C03568=1021.069,418.484,-159.354,174.058,50.310,160.418
C03569=1021.080,418.730,-159.402,174.072,50.312,160.420
C03570=1021.092,418.975,-159.450,174.087,50.313,160.423
C03571=1021.104,419.220,-159.498,174.100,50.315,160.426
C03572=1021.115,419.465,-159.546,174.115,50.316,160.429
C03573=1021.127,419.710,-159.594,174.129,50.318,160.432
C03574=1021.139,419.955,-159.641,174.143,50.320,160.435
C03575=1021.150,420.201,-159.690,174.158,50.321,160.438
C03576=1021.161,420.446,-159.737,174.171,50.323,160.441
C03577=1021.173,420.691,-159.786,174.186,50.325,160.444
C03578=1021.185,420.936,-159.834,174.201,50.326,160.446
C03579=1021.197,421.181,-159.882,174.215,50.328,160.449
C03580=1021.208,421.427,-159.930,174.229,50.330,160.453
C03581=1021.220,421.671,-159.979,174.244,50.331,160.455
C03582=1021.231,421.916,-160.027,174.259,50.333,160.458
C03583=1021.243,422.161,-160.076,174.273,50.335,160.461
C03584=1021.255,422.406,-160.125,174.287,50.337,160.464
C03585=1021.267,422.652,-160.173,174.302,50.338,160.467
C03586=1021.279,422.896,-160.222,174.317,50.340,160.471
C03587=1021.290,423.141,-160.271,174.332,50.342,160.474
C03588=1021.302,423.386,-160.320,174.347,50.344,160.477
C03589=1021.314,423.631,-160.368,174.362,50.346,160.480
C03590=1021.326,423.877,-160.417,174.377,50.348,160.483
C03591=1021.338,424.121,-160.466,174.392,50.349,160.486
C03592=1021.350,424.365,-160.515,174.407,50.351,160.489
C03593=1021.363,424.610,-160.564,174.422,50.354,160.492
C03594=1021.375,424.856,-160.613,174.437,50.355,160.495
C03595=1021.386,425.101,-160.662,174.452,50.358,160.499
C03596=1021.399,425.346,-160.711,174.467,50.359,160.502
C03597=1021.411,425.591,-160.761,174.482,50.362,160.505
C03598=1021.423,425.835,-160.810,174.498,50.363,160.508
C03599=1021.435,426.081,-160.860,174.513,50.365,160.511
C03600=1021.446,426.325,-160.909,174.529,50.367,160.515
C03601=1021.459,426.570,-160.958,174.544,50.370,160.518
C03602=1021.471,426.810,-161.007,174.559,50.371,160.521
C03603=1021.483,427.050,-161.056,174.574,50.374,160.524
C03604=1021.495,427.290,-161.104,174.589,50.376,160.528
C03605=1021.507,427.530,-161.153,174.605,50.378,160.531
C03606=1021.519,427.770,-161.202,174.620,50.379,160.534
C03607=1021.531,428.009,-161.252,174.636,50.382,160.537
C03608=1021.544,428.249,-161.300,174.651,50.384,160.541
C03609=1021.555,428.488,-161.349,174.666,50.386,160.544
C03610=1021.567,428.733,-161.399,174.682,50.388,160.547
C03611=1021.580,428.978,-161.449,174.698,50.391,160.551
C03612=1021.592,429.223,-161.499,174.714,50.393,160.554
C03613=1021.605,429.467,-161.549,174.730,50.395,160.557
C03614=1021.618,429.712,-161.599,174.746,50.397,160.561
C03615=1021.630,429.956,-161.649,174.762,50.399,160.564
C03616=1021.643,430.202,-161.700,174.778,50.402,160.568
C03617=1021.655,430.446,-161.751,174.795,50.404,160.571
C03618=1021.272,428.491,-161.685,174.655,50.455,160.562
C03619=1021.261,428.264,-161.639,174.641,50.453,160.559
C03620=1021.250,428.037,-161.592,174.626,50.451,160.556
C03621=1021.238,427.810,-161.547,174.611,50.449,160.553
C03622=1021.227,427.582,-161.500,174.597,50.447,160.550
C03623=1021.216,427.356,-161.454,174.582,50.445,160.547
C03624=1021.204,427.128,-161.408,174.567,50.444,160.544
C03625=1021.193,426.901,-161.361,174.553,50.442,160.541
C03626=1021.182,426.673,-161.315,174.539,50.440,160.538
C03627=1021.169,426.429,-161.267,174.523,50.438,160.534
C03628=1021.157,426.184,-161.216,174.508,50.436,160.531
C03629=1021.146,425.939,-161.167,174.492,50.434,160.528
C03630=1021.133,425.695,-161.117,174.477,50.432,160.525
C03631=1021.121,425.449,-161.068,174.462,50.430,160.522
C03632=1021.109,425.205,-161.020,174.447,50.428,160.518
C03633=1021.097,424.959,-160.970,174.431,50.426,160.515
C03634=1021.085,424.714,-160.921,174.416,50.425,160.512
C03635=1021.073,424.470,-160.872,174.401,50.423,160.509
C03636=1021.061,424.224,-160.822,174.386,50.421,160.506
C03637=1021.049,423.980,-160.774,174.371,50.419,160.503
C03638=1021.037,423.735,-160.724,174.356,50.417,160.500
C03639=1021.025,423.490,-160.677,174.341,50.416,160.496
C03640=1021.013,423.245,-160.628,174.326,50.414,160.493
C03641=1021.001,422.999,-160.578,174.311,50.412,160.490
C03642=1020.989,422.755,-160.530,174.297,50.410,160.487
C03643=1020.978,422.510,-160.481,174.282,50.409,160.484
C03644=1020.966,422.265,-160.433,174.267,50.407,160.481
C03645=1020.954,422.020,-160.384,174.252,50.406,160.478
C03646=1020.942,421.775,-160.336,174.237,50.404,160.475
C03647=1020.931,421.530,-160.287,174.223,50.402,160.472
C03648=1020.920,421.285,-160.239,174.209,50.400,160.469
C03649=1020.907,421.040,-160.190,174.194,50.399,160.466
C03650=1020.895,420.794,-160.142,174.179,50.397,160.463
C03651=1020.884,420.549,-160.094,174.165,50.396,160.460
C03652=1020.872,420.304,-160.046,174.150,50.395,160.458
C03653=1020.861,420.059,-159.998,174.136,50.393,160.455
C03654=1020.849,419.814,-159.950,174.122,50.391,160.452
C03655=1020.837,419.569,-159.902,174.108,50.390,160.449
C03656=1020.826,419.324,-159.854,174.094,50.388,160.446
C03657=1020.814,419.079,-159.806,174.079,50.387,160.443
C03658=1020.803,418.833,-159.759,174.065,50.386,160.440
C03659=1020.791,418.588,-159.711,174.051,50.384,160.437
C03660=1020.780,418.343,-159.663,174.037,50.383,160.435
C03661=1020.768,418.098,-159.616,174.023,50.381,160.432
C03662=1020.757,417.853,-159.567,174.009,50.380,160.429
C03663=1020.746,417.607,-159.520,173.995,50.378,160.426
C03664=1020.734,417.362,-159.473,173.981,50.377,160.423
C03665=1020.723,417.117,-159.425,173.967,50.376,160.421
C03666=1020.712,416.872,-159.378,173.954,50.374,160.418
C03667=1020.701,416.626,-159.329,173.940,50.373,160.415
C03668=1020.690,416.381,-159.283,173.926,50.372,160.412
C03669=1020.678,416.136,-159.235,173.913,50.370,160.410
C03670=1020.667,415.890,-159.187,173.898,50.369,160.407
C03671=1020.656,415.645,-159.141,173.885,50.368,160.404
C03672=1020.644,415.400,-159.093,173.872,50.366,160.401
C03673=1020.634,415.155,-159.046,173.858,50.365,160.399
C03674=1020.623,414.909,-158.999,173.844,50.364,160.396
C03675=1020.612,414.664,-158.952,173.831,50.363,160.394
C03676=1020.600,414.419,-158.905,173.818,50.362,160.391
C03677=1020.589,414.174,-158.859,173.803,50.360,160.388
C03678=1020.578,413.928,-158.812,173.790,50.359,160.386
C03679=1020.568,413.683,-158.765,173.777,50.358,160.383
C03680=1020.556,413.437,-158.718,173.764,50.357,160.381
C03681=1020.545,413.192,-158.672,173.751,50.356,160.378
C03682=1020.535,412.947,-158.625,173.738,50.355,160.375
C03683=1020.519,412.599,-158.559,173.719,50.353,160.372
C03684=1020.503,412.251,-158.493,173.700,50.352,160.368
C03685=1020.488,411.903,-158.427,173.682,50.351,160.365
C03686=1020.472,411.556,-158.361,173.663,50.349,160.361
C03687=1020.461,411.311,-158.315,173.651,50.348,160.359
C03688=1020.451,411.065,-158.269,173.637,50.347,160.356
C03689=1020.440,410.820,-158.223,173.624,50.346,160.353
C03690=1020.430,410.574,-158.176,173.611,50.345,160.351
C03691=1020.419,410.329,-158.130,173.599,50.344,160.349
C03692=1020.409,410.083,-158.084,173.586,50.343,160.346
C03693=1020.398,409.838,-158.037,173.573,50.342,160.344
C03694=1020.387,409.592,-157.991,173.561,50.341,160.341
C03695=1020.376,409.347,-157.945,173.548,50.340,160.339
C03696=1020.366,409.101,-157.900,173.535,50.340,160.336
C03697=1020.355,408.856,-157.854,173.523,50.338,160.334
C03698=1020.345,408.610,-157.808,173.510,50.338,160.332
C03699=1020.334,408.365,-157.762,173.497,50.337,160.329
C03700=1020.323,408.119,-157.716,173.484,50.336,160.327
C03701=1020.312,407.873,-157.671,173.473,50.335,160.324
C03702=1020.302,407.627,-157.625,173.460,50.335,160.322
C03703=1020.291,407.382,-157.579,173.447,50.334,160.320
C03704=1020.281,407.137,-157.534,173.434,50.334,160.317
C03705=1020.271,406.891,-157.489,173.423,50.333,160.315
C03706=1020.259,406.645,-157.443,173.410,50.332,160.313
C03707=1020.249,406.399,-157.398,173.398,50.331,160.311
C03708=1020.239,406.154,-157.353,173.386,50.331,160.308
C03709=1020.229,405.908,-157.308,173.373,50.330,160.306
C03710=1020.217,405.663,-157.262,173.361,50.329,160.304
C03711=1020.208,405.417,-157.217,173.349,50.329,160.301
C03712=1020.197,405.172,-157.171,173.337,50.328,160.299
C03713=1020.187,404.926,-157.127,173.324,50.327,160.297
C03714=1020.177,404.680,-157.081,173.313,50.327,160.295
C03715=1020.166,404.435,-157.037,173.300,50.326,160.292
C03716=1020.156,404.189,-156.991,173.288,50.325,160.290
C03717=1020.146,403.944,-156.947,173.276,50.325,160.288
C03718=1020.136,403.697,-156.901,173.264,50.324,160.286
C03719=1020.125,403.452,-156.857,173.253,50.324,160.284
C03720=1020.115,403.206,-156.812,173.240,50.323,160.281
C03721=1020.105,402.961,-156.767,173.229,50.323,160.279
C03722=1020.096,402.715,-156.722,173.216,50.323,160.277
C03723=1020.085,402.469,-156.677,173.205,50.322,160.275
C03724=1020.075,402.224,-156.633,173.193,50.321,160.273
C03725=1020.065,401.978,-156.588,173.181,50.321,160.271
C03726=1020.055,401.733,-156.543,173.169,50.320,160.268
C03727=1020.045,401.486,-156.498,173.158,50.320,160.266
C03728=1020.035,401.241,-156.454,173.147,50.320,160.264
C03729=1020.025,400.995,-156.410,173.134,50.320,160.262
C03730=1020.016,400.750,-156.365,173.123,50.319,160.260
C03731=1020.006,400.503,-156.321,173.111,50.318,160.258
C03732=1019.995,400.257,-156.276,173.100,50.318,160.256
C03733=1019.986,400.011,-156.232,173.088,50.318,160.254
C03734=1019.976,399.766,-156.187,173.076,50.318,160.252
C03735=1019.966,399.520,-156.144,173.065,50.317,160.250
C03736=1019.956,399.275,-156.099,173.054,50.317,160.248
C03737=1019.946,399.029,-156.055,173.042,50.316,160.246
C03738=1019.937,398.783,-156.011,173.031,50.316,160.244
C03739=1019.927,398.537,-155.966,173.020,50.316,160.242
C03740=1019.917,398.291,-155.923,173.008,50.316,160.240
C03741=1019.907,398.045,-155.879,172.997,50.316,160.238
C03742=1019.897,397.799,-155.835,172.985,50.316,160.236
C03743=1019.885,397.475,-155.777,172.971,50.316,160.233
C03744=1019.872,397.150,-155.720,172.955,50.315,160.231
C03745=1019.858,396.825,-155.662,172.941,50.315,160.228
C03746=1019.846,396.500,-155.604,172.926,50.315,160.226
C03747=1019.836,396.254,-155.560,172.915,50.315,160.224
C03748=1019.826,396.009,-155.517,172.904,50.315,160.222
C03749=1019.816,395.762,-155.473,172.892,50.315,160.220
C03750=1019.807,395.516,-155.430,172.882,50.315,160.218
C03751=1019.798,395.271,-155.386,172.871,50.314,160.216
C03752=1019.788,395.025,-155.343,172.860,50.314,160.214
C03753=1019.777,394.779,-155.299,172.849,50.315,160.212
C03754=1019.768,394.532,-155.256,172.838,50.315,160.211
C03755=1019.759,394.287,-155.213,172.827,50.314,160.208
C03756=1019.749,394.041,-155.170,172.816,50.314,160.207
C03757=1019.740,393.794,-155.126,172.805,50.315,160.205
C03758=1019.730,393.549,-155.083,172.794,50.315,160.203
C03759=1019.721,393.303,-155.039,172.783,50.315,160.201
C03760=1019.711,393.056,-154.997,172.773,50.315,160.200
C03761=1019.702,392.810,-154.954,172.763,50.315,160.198
C03762=1019.692,392.564,-154.910,172.751,50.315,160.196
C03763=1019.683,392.318,-154.868,172.740,50.315,160.194
C03764=1019.673,392.072,-154.825,172.730,50.316,160.192
C03765=1019.664,391.826,-154.782,172.720,50.315,160.191
C03766=1019.655,391.580,-154.739,172.709,50.316,160.189
C03767=1019.645,391.334,-154.696,172.698,50.316,160.187
C03768=1019.636,391.088,-154.653,172.687,50.316,160.185
C03769=1019.626,390.842,-154.611,172.677,50.316,160.183
C03770=1019.616,390.596,-154.568,172.667,50.317,160.182
C03771=1019.608,390.350,-154.525,172.656,50.317,160.180
C03772=1019.599,390.103,-154.483,172.645,50.317,160.178
C03773=1019.589,389.857,-154.440,172.635,50.317,160.177
C03774=1019.580,389.611,-154.398,172.624,50.318,160.175
C03775=1019.571,389.365,-154.355,172.614,50.317,160.173
C03776=1019.562,389.119,-154.312,172.604,50.318,160.171
C03777=1019.552,388.873,-154.270,172.593,50.318,160.170
C03778=1019.543,388.627,-154.228,172.583,50.319,160.168
C03779=1019.534,388.380,-154.185,172.572,50.319,160.166
C03780=1019.524,388.134,-154.143,172.562,50.320,160.165
C03781=1019.515,387.888,-154.101,172.552,50.319,160.163
C03782=1019.506,387.642,-154.058,172.541,50.320,160.161
C03783=1019.497,387.395,-154.016,172.532,50.321,160.160
C03784=1019.488,387.149,-153.973,172.521,50.321,160.158
C03785=1019.479,386.903,-153.932,172.511,50.321,160.156
C03786=1019.470,386.656,-153.890,172.501,50.322,160.155
C03787=1019.461,386.411,-153.847,172.490,50.323,160.153
C03788=1019.452,386.164,-153.806,172.481,50.323,160.152
C03789=1019.443,385.918,-153.764,172.470,50.323,160.150
C03790=1019.434,385.672,-153.722,172.460,50.324,160.148
C03791=1019.425,385.426,-153.680,172.451,50.324,160.147
C03792=1019.416,385.179,-153.638,172.440,50.325,160.145
C03793=1019.407,384.932,-153.596,172.431,50.325,160.144
C03794=1019.397,384.686,-153.555,172.420,50.326,160.142
C03795=1019.388,384.440,-153.513,172.410,50.326,160.141
C03796=1019.379,384.194,-153.472,172.400,50.327,160.139
C03797=1019.370,383.947,-153.430,172.391,50.328,160.138
C03798=1019.361,383.701,-153.388,172.380,50.329,160.136
C03799=1019.351,383.455,-153.347,172.371,50.329,160.135
C03800=1019.343,383.209,-153.306,172.360,50.330,160.133
C03801=1019.335,382.962,-153.265,172.351,50.330,160.132
C03802=1019.326,382.716,-153.223,172.341,50.331,160.130
C03803=1019.314,382.429,-153.174,172.329,50.332,160.128
C03804=1019.304,382.141,-153.127,172.318,50.333,160.127
C03805=1019.294,381.854,-153.079,172.306,50.334,160.125
C03806=1019.283,381.567,-153.030,172.296,50.335,160.123
C03807=1019.275,381.321,-152.989,172.285,50.336,160.122
C03808=1019.266,381.074,-152.948,172.276,50.336,160.120
C03809=1019.257,380.828,-152.906,172.267,50.337,160.119
C03810=1019.248,380.581,-152.865,172.256,50.338,160.117
C03811=1019.239,380.335,-152.824,172.247,50.339,160.116
C03812=1019.231,380.088,-152.783,172.238,50.340,160.115
C03813=1019.222,379.841,-152.742,172.228,50.340,160.113
C03814=1019.214,379.596,-152.701,172.218,50.341,160.112
C03815=1019.205,379.349,-152.660,172.208,50.342,160.110
C03816=1019.196,379.102,-152.620,172.199,50.343,160.109
C03817=1019.188,378.857,-152.578,172.190,50.344,160.108
C03818=1019.179,378.610,-152.537,172.180,50.344,160.106
C03819=1019.171,378.363,-152.497,172.170,50.345,160.105
C03820=1019.162,378.117,-152.455,172.161,50.346,160.103
C03821=1019.153,377.871,-152.415,172.152,50.347,160.102
C03822=1019.145,377.624,-152.374,172.143,50.348,160.101
C03823=1019.137,377.378,-152.333,172.133,50.349,160.099
C03824=1019.128,377.131,-152.292,172.123,50.350,160.098
C03825=1019.119,376.885,-152.252,172.114,50.351,160.097
C03826=1019.110,376.638,-152.211,172.105,50.352,160.095
C03827=1019.102,376.391,-152.170,172.096,50.353,160.094
C03828=1019.094,376.144,-152.129,172.087,50.354,160.093
C03829=1019.086,375.898,-152.089,172.077,50.355,160.091
C03830=1019.076,375.651,-152.048,172.068,50.356,160.090
C03831=1019.068,375.405,-152.008,172.059,50.357,160.089
C03832=1019.060,375.159,-151.968,172.050,50.358,160.087
C03833=1019.051,374.912,-151.928,172.040,50.359,160.086
C03834=1019.043,374.666,-151.887,172.031,50.361,160.085
C03835=1019.034,374.418,-151.848,172.022,50.362,160.084
C03836=1019.025,374.172,-151.807,172.013,50.363,160.082
C03837=1019.017,373.925,-151.768,172.003,50.364,160.081
C03838=1019.009,373.679,-151.727,171.995,50.365,160.080
C03839=1019.000,373.432,-151.687,171.986,50.366,160.079
C03840=1018.991,373.186,-151.647,171.976,50.367,160.077
C03841=1018.983,372.939,-151.608,171.968,50.369,160.076
C03842=1018.974,372.692,-151.567,171.958,50.370,160.075
C03843=1018.966,372.445,-151.527,171.950,50.372,160.074
C03844=1018.958,372.199,-151.487,171.940,50.372,160.072
C03845=1018.950,371.953,-151.447,171.932,50.374,160.071
C03846=1018.941,371.706,-151.408,171.923,50.375,160.070
C03847=1018.933,371.460,-151.367,171.914,50.377,160.069
C03848=1018.924,371.212,-151.328,171.905,50.378,160.068
C03849=1018.916,370.966,-151.288,171.896,50.379,160.067
C03850=1018.908,370.719,-151.248,171.887,50.380,160.065
C03851=1018.899,370.473,-151.208,171.878,50.382,160.064
C03852=1018.892,370.226,-151.168,171.869,50.383,160.063
C03853=1018.883,369.979,-151.129,171.860,50.384,160.062
C03854=1018.876,369.732,-151.089,171.851,50.386,160.061
C03855=1018.867,369.486,-151.050,171.842,50.387,160.059
C03856=1018.859,369.239,-151.010,171.834,50.388,160.058
C03857=1018.851,368.992,-150.971,171.825,50.390,160.057
C03858=1018.842,368.746,-150.931,171.817,50.391,160.056
C03859=1018.835,368.499,-150.891,171.808,50.393,160.055
C03860=1018.826,368.252,-150.852,171.799,50.394,160.054
C03861=1018.819,368.005,-150.812,171.790,50.395,160.053
C03862=1018.810,367.759,-150.773,171.781,50.397,160.051
C03863=1018.801,367.494,-150.731,171.772,50.398,160.050
C03864=1018.793,367.229,-150.689,171.763,50.400,160.049
C03865=1018.784,366.963,-150.647,171.754,50.402,160.048
C03866=1018.775,366.699,-150.604,171.745,50.404,160.047
C03867=1018.767,366.452,-150.566,171.736,50.405,160.046
C03868=1018.759,366.205,-150.527,171.727,50.407,160.045
C03869=1018.750,365.958,-150.488,171.719,50.408,160.044
C03870=1018.743,365.712,-150.449,171.710,50.410,160.043
C03871=1018.734,365.465,-150.410,171.701,50.411,160.041
C03872=1018.727,365.218,-150.370,171.693,50.413,160.040
C03873=1018.719,364.971,-150.332,171.685,50.415,160.040
C03874=1018.710,364.724,-150.293,171.676,50.416,160.038
C03875=1018.703,364.477,-150.254,171.667,50.418,160.037
C03876=1018.694,364.230,-150.216,171.659,50.420,160.036
C03877=1018.686,363.984,-150.176,171.651,50.421,160.035
C03878=1018.678,363.737,-150.138,171.642,50.423,160.034
C03879=1018.670,363.490,-150.100,171.634,50.425,160.033
C03880=1018.662,363.243,-150.060,171.625,50.427,160.032
C03881=1018.654,362.997,-150.022,171.617,50.428,160.031
C03882=1018.647,362.749,-149.983,171.609,50.430,160.030
C03883=1018.639,362.502,-149.944,171.600,50.432,160.029
C03884=1018.631,362.256,-149.906,171.591,50.433,160.028
C03885=1018.623,362.009,-149.867,171.584,50.435,160.027
C03886=1018.615,361.762,-149.828,171.575,50.437,160.026
C03887=1018.607,361.515,-149.790,171.567,50.439,160.025
C03888=1018.599,361.268,-149.751,171.560,50.441,160.025
C03889=1018.591,361.022,-149.713,171.551,50.442,160.023
C03890=1018.583,360.774,-149.674,171.542,50.445,160.023
C03891=1018.577,360.563,-149.641,171.536,50.445,160.022
C03892=1018.571,360.352,-149.609,171.528,50.447,160.021
C03893=1018.564,360.142,-149.575,171.522,50.449,160.020
C03894=1018.557,359.931,-149.543,171.514,50.451,160.019
C03895=1018.550,359.720,-149.510,171.508,50.452,160.019
C03896=1018.544,359.509,-149.478,171.501,50.454,160.018
C03897=1018.538,359.299,-149.445,171.494,50.455,160.017
C03898=1018.531,359.088,-149.413,171.487,50.457,160.016
C03899=1018.523,358.841,-149.375,171.478,50.459,160.015
C03900=1018.515,358.595,-149.336,171.471,50.461,160.014
C03901=1018.507,358.347,-149.298,171.462,50.463,160.013
C03902=1018.500,358.100,-149.260,171.455,50.465,160.013
C03903=1018.492,357.853,-149.222,171.446,50.467,160.012
C03904=1018.484,357.606,-149.184,171.438,50.469,160.011
C03905=1018.476,357.360,-149.146,171.431,50.471,160.010
C03906=1018.468,357.112,-149.108,171.422,50.473,160.009
C03907=1018.461,356.865,-149.070,171.414,50.475,160.008
C03908=1018.453,356.618,-149.033,171.406,50.477,160.007
C03909=1018.445,356.371,-148.994,171.398,50.479,160.006
C03910=1018.437,356.124,-148.957,171.391,50.481,160.006
C03911=1018.430,355.877,-148.920,171.382,50.483,160.005
C03912=1018.423,355.631,-148.881,171.374,50.485,160.004
C03913=1018.415,355.383,-148.843,171.366,50.487,160.003
C03914=1018.407,355.136,-148.807,171.358,50.490,160.002
C03915=1018.399,354.889,-148.768,171.351,50.492,160.001
C03916=1018.392,354.642,-148.731,171.343,50.494,160.001
C03917=1018.385,354.395,-148.693,171.335,50.496,160.000
C03918=1018.376,354.148,-148.656,171.327,50.498,159.999
C03919=1018.369,353.900,-148.618,171.320,50.501,159.998
C03920=1018.361,353.654,-148.580,171.311,50.503,159.997
C03921=1018.354,353.407,-148.543,171.304,50.505,159.997
C03922=1018.346,353.160,-148.506,171.296,50.508,159.996
C03923=1018.336,352.830,-148.457,171.286,50.510,159.995
C03924=1018.326,352.500,-148.406,171.275,50.513,159.994
C03925=1018.315,352.170,-148.356,171.265,50.516,159.993
C03926=1018.305,351.840,-148.306,171.255,50.520,159.992
C03927=1018.298,351.592,-148.270,171.246,50.522,159.991
C03928=1018.290,351.346,-148.233,171.239,50.524,159.990
C03929=1018.283,351.098,-148.195,171.231,50.527,159.989
C03930=1018.276,350.851,-148.158,171.224,50.529,159.989
C03931=1018.268,350.604,-148.121,171.216,50.531,159.988
C03932=1018.261,350.357,-148.084,171.209,50.534,159.987
C03933=1018.253,350.110,-148.047,171.200,50.536,159.986
C03934=1018.246,349.863,-148.009,171.193,50.538,159.986
C03935=1018.238,349.616,-147.973,171.185,50.541,159.985
C03936=1018.231,349.368,-147.936,171.178,50.543,159.984
C03937=1018.223,349.121,-147.898,171.171,50.545,159.984
C03938=1018.216,348.874,-147.862,171.163,50.548,159.983
C03939=1018.209,348.627,-147.825,171.156,50.551,159.982
C03940=1018.201,348.380,-147.788,171.147,50.553,159.981
C03941=1018.194,348.133,-147.751,171.140,50.555,159.981
C03942=1018.186,347.886,-147.714,171.132,50.558,159.980
C03943=1018.179,347.638,-147.677,171.125,50.561,159.980
C03944=1018.171,347.391,-147.640,171.118,50.563,159.979
C03945=1018.165,347.144,-147.604,171.110,50.565,159.978
C03946=1018.157,346.897,-147.567,171.103,50.568,159.977
C03947=1018.150,346.650,-147.530,171.095,50.571,159.977
C03948=1018.142,346.402,-147.494,171.088,50.573,159.976
C03949=1018.135,346.155,-147.458,171.080,50.576,159.975
C03950=1018.128,345.908,-147.421,171.073,50.578,159.975
C03951=1018.120,345.661,-147.384,171.066,50.581,159.974
C03952=1018.113,345.413,-147.348,171.058,50.584,159.973
C03953=1018.106,345.166,-147.312,171.051,50.586,159.973
C03954=1018.099,344.919,-147.275,171.043,50.589,159.972
C03955=1018.091,344.672,-147.239,171.036,50.592,159.972
C03956=1018.083,344.425,-147.202,171.029,50.594,159.971
C03957=1018.077,344.178,-147.166,171.021,50.597,159.970
C03958=1018.069,343.930,-147.130,171.014,50.600,159.970
C03959=1018.061,343.683,-147.093,171.006,50.603,159.969
C03960=1018.055,343.436,-147.057,170.999,50.605,159.969
C03961=1018.047,343.188,-147.021,170.992,50.608,159.968
C03962=1018.040,342.941,-146.985,170.984,50.611,159.967
C03963=1018.033,342.694,-146.948,170.977,50.613,159.967
C03964=1018.026,342.446,-146.912,170.970,50.616,159.966
C03965=1018.018,342.199,-146.876,170.963,50.619,159.966
C03966=1018.011,341.951,-146.841,170.956,50.622,159.965
C03967=1018.005,341.704,-146.804,170.949,50.624,159.964
C03968=1017.997,341.457,-146.768,170.941,50.628,159.964
C03969=1017.990,341.210,-146.732,170.934,50.630,159.963
C03970=1017.982,340.963,-146.696,170.927,50.633,159.963
C03971=1017.976,340.715,-146.661,170.920,50.636,159.962
C03972=1017.969,340.468,-146.624,170.913,50.639,159.962
C03973=1017.962,340.221,-146.588,170.906,50.642,159.961
C03974=1017.954,339.973,-146.552,170.898,50.645,159.961
C03975=1017.947,339.726,-146.517,170.891,50.648,159.960
C03976=1017.939,339.479,-146.480,170.884,50.650,159.960
C03977=1017.933,339.231,-146.445,170.877,50.654,159.959
C03978=1017.926,338.984,-146.409,170.870,50.656,159.958
C03979=1017.919,338.737,-146.373,170.863,50.659,159.958
C03980=1017.912,338.489,-146.338,170.855,50.663,159.958
C03981=1017.905,338.241,-146.302,170.848,50.665,159.957
C03982=1017.897,337.995,-146.266,170.842,50.668,159.956
C03983=1017.890,337.735,-146.229,170.834,50.672,159.956
C03984=1017.883,337.474,-146.192,170.826,50.674,159.955
C03985=1017.875,337.214,-146.155,170.819,50.678,159.955
C03986=1017.867,336.953,-146.117,170.812,50.681,159.954
C03987=1017.860,336.706,-146.082,170.805,50.684,159.954
C03988=1017.853,336.459,-146.047,170.798,50.688,159.953
C03989=1017.846,336.211,-146.011,170.791,50.690,159.953
C03990=1017.839,335.964,-145.975,170.784,50.693,159.952
C03991=1017.832,335.717,-145.940,170.776,50.697,159.952
C03992=1017.825,335.469,-145.905,170.770,50.700,159.952
C03993=1017.818,335.221,-145.869,170.763,50.703,159.951
C03994=1017.811,334.974,-145.834,170.756,50.706,159.951
C03995=1017.804,334.727,-145.798,170.749,50.709,159.950
C03996=1017.797,334.480,-145.763,170.742,50.713,159.950
C03997=1017.790,334.232,-145.728,170.736,50.716,159.949
C03998=1017.783,333.984,-145.693,170.729,50.719,159.949
C03999=1017.777,333.737,-145.658,170.721,50.722,159.949
C04000=1017.770,333.490,-145.622,170.715,50.725,159.948
C04001=1017.763,333.242,-145.587,170.708,50.728,159.948
C04002=1017.756,332.995,-145.552,170.702,50.732,159.947
C04003=1017.749,332.747,-145.517,170.694,50.735,159.947
C04004=1017.741,332.500,-145.482,170.687,50.738,159.946
C04005=1017.735,332.252,-145.447,170.681,50.741,159.946
C04006=1017.728,332.005,-145.412,170.674,50.744,159.946
C04007=1017.721,331.757,-145.377,170.666,50.748,159.945
C04008=1017.714,331.510,-145.343,170.660,50.752,159.945
C04009=1017.707,331.263,-145.308,170.654,50.755,159.944
C04010=1017.700,331.015,-145.273,170.647,50.758,159.944
C04011=1017.693,330.768,-145.239,170.639,50.761,159.944
C04012=1017.686,330.520,-145.204,170.633,50.765,159.943
C04013=1017.680,330.273,-145.169,170.626,50.768,159.943
C04014=1017.672,330.025,-145.135,170.620,50.771,159.943
C04015=1017.666,329.778,-145.100,170.613,50.775,159.942
C04016=1017.659,329.530,-145.064,170.606,50.779,159.942
C04017=1017.652,329.282,-145.030,170.599,50.782,159.941
C04018=1017.645,329.035,-144.995,170.593,50.785,159.941
C04019=1017.638,328.787,-144.961,170.586,50.789,159.941
C04020=1017.632,328.540,-144.926,170.579,50.792,159.940
C04021=1017.624,328.292,-144.892,170.573,50.796,159.940
C04022=1017.618,328.045,-144.857,170.566,50.799,159.940
C04023=1017.611,327.797,-144.823,170.560,50.803,159.939
C04024=1017.604,327.550,-144.788,170.552,50.806,159.939
C04025=1017.598,327.303,-144.754,170.546,50.810,159.939
C04026=1017.591,327.055,-144.719,170.539,50.813,159.938
C04027=1017.584,326.808,-144.685,170.533,50.817,159.938
C04028=1017.577,326.560,-144.651,170.526,50.820,159.938
C04029=1017.571,326.312,-144.615,170.519,50.824,159.937
C04030=1017.563,326.065,-144.582,170.513,50.828,159.937
C04031=1017.557,325.818,-144.548,170.506,50.831,159.937
C04032=1017.550,325.570,-144.514,170.500,50.835,159.937
C04033=1017.543,325.322,-144.480,170.493,50.839,159.936
C04034=1017.536,325.075,-144.445,170.487,50.843,159.936
C04035=1017.529,324.827,-144.412,170.480,50.846,159.936
C04036=1017.522,324.579,-144.377,170.474,50.849,159.935
C04037=1017.515,324.332,-144.344,170.467,50.854,159.935
C04038=1017.508,324.085,-144.310,170.460,50.857,159.935
C04039=1017.501,323.837,-144.276,170.454,50.861,159.935
C04040=1017.495,323.589,-144.242,170.448,50.865,159.935
C04041=1017.488,323.342,-144.208,170.441,50.869,159.934
C04042=1017.481,323.094,-144.175,170.434,50.872,159.934
C04043=1017.474,322.829,-144.138,170.427,50.877,159.934
C04044=1017.466,322.565,-144.102,170.421,50.881,159.934
C04045=1017.459,322.300,-144.066,170.414,50.885,159.933
C04046=1017.452,322.035,-144.030,170.407,50.889,159.933
C04047=1017.445,321.788,-143.996,170.400,50.893,159.933
C04048=1017.438,321.540,-143.963,170.394,50.896,159.933
C04049=1017.431,321.292,-143.929,170.388,50.900,159.932
C04050=1017.425,321.045,-143.895,170.381,50.904,159.932
C04051=1017.418,320.798,-143.861,170.375,50.908,159.932
C04052=1017.412,320.550,-143.829,170.368,50.912,159.932
C04053=1017.405,320.302,-143.795,170.362,50.916,159.931
C04054=1017.397,320.055,-143.761,170.356,50.919,159.931
C04055=1017.392,319.807,-143.727,170.349,50.924,159.931
C04056=1017.385,319.559,-143.694,170.342,50.927,159.931
C04057=1017.378,319.312,-143.660,170.337,50.932,159.931
C04058=1017.371,319.064,-143.627,170.330,50.936,159.930
C04059=1017.365,318.816,-143.593,170.324,50.939,159.930
C04060=1017.358,318.569,-143.559,170.317,50.943,159.930
C04061=1017.352,318.321,-143.527,170.311,50.947,159.930
C04062=1017.345,318.074,-143.493,170.305,50.952,159.930
C04063=1017.339,317.826,-143.459,170.299,50.955,159.930
C04064=1017.332,317.578,-143.426,170.292,50.959,159.929
C04065=1017.325,317.331,-143.392,170.286,50.963,159.929
C04066=1017.318,317.083,-143.359,170.279,50.968,159.929
C04067=1017.312,316.836,-143.326,170.273,50.972,159.929
C04068=1017.306,316.588,-143.292,170.267,50.975,159.929
C04069=1017.299,316.340,-143.259,170.261,50.980,159.929
C04070=1017.293,316.093,-143.226,170.255,50.984,159.928
C04071=1017.286,315.844,-143.193,170.249,50.987,159.928
C04072=1017.280,315.597,-143.159,170.242,50.992,159.928
C04073=1017.274,315.349,-143.126,170.236,50.996,159.928
C04074=1017.267,315.101,-143.093,170.230,51.000,159.928
C04075=1017.260,314.854,-143.059,170.224,51.004,159.928
C04076=1017.254,314.607,-143.026,170.217,51.008,159.927
C04077=1017.248,314.359,-142.993,170.212,51.012,159.927
C04078=1017.241,314.111,-142.959,170.205,51.016,159.927
C04079=1017.235,313.863,-142.927,170.198,51.021,159.927
C04080=1017.229,313.616,-142.894,170.192,51.025,159.927
C04081=1017.221,313.368,-142.860,170.186,51.029,159.927
C04082=1017.216,313.120,-142.827,170.180,51.033,159.927
C04083=1017.209,312.873,-142.794,170.174,51.037,159.927
C04084=1017.203,312.625,-142.761,170.169,51.042,159.927
C04085=1017.197,312.377,-142.728,170.162,51.046,159.926
C04086=1017.190,312.130,-142.695,170.157,51.050,159.926
C04087=1017.184,311.882,-142.661,170.150,51.054,159.926
C04088=1017.178,311.634,-142.629,170.143,51.059,159.926
C04089=1017.172,311.387,-142.596,170.138,51.063,159.926
C04090=1017.165,311.139,-142.563,170.131,51.067,159.926
C04091=1017.159,310.891,-142.530,170.126,51.071,159.926
C04092=1017.153,310.644,-142.497,170.120,51.076,159.926
C04093=1017.147,310.395,-142.464,170.114,51.080,159.926
C04094=1017.140,310.148,-142.431,170.108,51.084,159.926
C04095=1017.134,309.900,-142.398,170.102,51.089,159.926
C04096=1017.128,309.652,-142.366,170.096,51.092,159.925
C04097=1017.121,309.405,-142.333,170.089,51.097,159.925
C04098=1017.115,309.157,-142.300,170.083,51.102,159.925
C04099=1017.108,308.909,-142.269,170.077,51.106,159.925
C04100=1017.102,308.662,-142.236,170.071,51.110,159.925
C04101=1017.095,308.415,-142.204,170.066,51.115,159.925
C04102=1017.089,308.166,-142.172,170.059,51.120,159.925
C04103=1017.082,307.907,-142.138,170.053,51.125,159.925
C04104=1017.075,307.648,-142.104,170.047,51.130,159.925
C04105=1017.068,307.389,-142.071,170.041,51.134,159.925
C04106=1017.061,307.130,-142.037,170.034,51.139,159.925
C04107=1017.055,306.882,-142.005,170.028,51.143,159.925
C04108=1017.048,306.634,-141.972,170.022,51.148,159.925
C04109=1017.042,306.386,-141.940,170.017,51.153,159.925
C04110=1017.035,306.139,-141.908,170.010,51.158,159.925
C04111=1017.029,305.891,-141.876,170.004,51.162,159.925
C04112=1017.022,305.643,-141.844,169.998,51.167,159.925
C04113=1017.016,305.395,-141.812,169.993,51.171,159.925
C04114=1017.010,305.147,-141.780,169.987,51.176,159.925
C04115=1017.003,304.900,-141.748,169.980,51.181,159.925
C04116=1016.997,304.651,-141.716,169.975,51.186,159.925
C04117=1016.990,304.404,-141.684,169.969,51.190,159.925
C04118=1016.984,304.156,-141.652,169.963,51.195,159.925
C04119=1016.977,303.908,-141.620,169.958,51.200,159.925
C04120=1016.971,303.660,-141.588,169.951,51.204,159.925
C04121=1016.965,303.412,-141.555,169.945,51.209,159.925
C04122=1016.959,303.165,-141.524,169.940,51.214,159.925
C04123=1016.953,302.917,-141.492,169.934,51.218,159.925
C04124=1016.946,302.670,-141.460,169.928,51.223,159.925
C04125=1016.940,302.421,-141.428,169.921,51.228,159.926
C04126=1016.933,302.173,-141.397,169.916,51.233,159.926
C04127=1016.927,301.925,-141.365,169.910,51.238,159.926
C04128=1016.920,301.677,-141.333,169.904,51.243,159.926
C04129=1016.915,301.430,-141.302,169.899,51.247,159.926
C04130=1016.908,301.183,-141.269,169.893,51.252,159.926
C04131=1016.902,300.934,-141.237,169.886,51.257,159.926
C04132=1016.896,300.686,-141.205,169.881,51.262,159.926
C04133=1016.889,300.438,-141.174,169.875,51.267,159.926
C04134=1016.884,300.191,-141.142,169.870,51.272,159.926
C04135=1016.877,299.943,-141.111,169.864,51.276,159.926
C04136=1016.871,299.695,-141.079,169.859,51.281,159.926
C04137=1016.865,299.447,-141.047,169.852,51.286,159.926
C04138=1016.859,299.199,-141.016,169.846,51.291,159.926
C04139=1016.852,298.951,-140.984,169.841,51.296,159.927
C04140=1016.846,298.703,-140.952,169.835,51.301,159.927
C04141=1016.840,298.455,-140.921,169.830,51.306,159.927
C04142=1016.834,298.208,-140.889,169.824,51.311,159.927
C04143=1016.828,297.959,-140.857,169.818,51.316,159.927
C04144=1016.822,297.712,-140.826,169.812,51.321,159.927
C04145=1016.816,297.464,-140.794,169.806,51.326,159.927
C04146=1016.809,297.216,-140.763,169.801,51.331,159.927
C04147=1016.803,296.968,-140.731,169.796,51.336,159.927
C04148=1016.798,296.720,-140.700,169.790,51.340,159.927
C04149=1016.792,296.472,-140.668,169.783,51.346,159.927
C04150=1016.786,296.225,-140.637,169.778,51.351,159.928
C04151=1016.780,295.976,-140.605,169.772,51.356,159.928
C04152=1016.773,295.729,-140.574,169.767,51.361,159.928
C04153=1016.767,295.481,-140.542,169.761,51.366,159.928
C04154=1016.761,295.233,-140.511,169.756,51.371,159.928
C04155=1016.756,294.985,-140.480,169.751,51.376,159.928
C04156=1016.750,294.737,-140.448,169.744,51.381,159.928
C04157=1016.744,294.490,-140.417,169.738,51.386,159.928
C04158=1016.738,294.241,-140.385,169.733,51.391,159.929
C04159=1016.732,293.997,-140.354,169.728,51.396,159.929
C04160=1016.726,293.752,-140.324,169.722,51.402,159.929
C04161=1016.720,293.507,-140.293,169.716,51.406,159.929
C04162=1016.714,293.262,-140.261,169.711,51.411,159.929
C04163=1016.708,293.018,-140.231,169.706,51.416,159.929
C04164=1016.702,292.773,-140.200,169.700,51.422,159.930
C04165=1016.696,292.529,-140.170,169.695,51.427,159.930
C04166=1016.690,292.284,-140.139,169.689,51.432,159.930
C04167=1016.684,292.037,-140.108,169.683,51.437,159.930
C04168=1016.678,291.789,-140.078,169.678,51.443,159.930
C04169=1016.672,291.540,-140.046,169.672,51.448,159.930
C04170=1016.666,291.293,-140.015,169.667,51.453,159.931
C04171=1016.660,291.044,-139.984,169.662,51.459,159.931
C04172=1016.654,290.796,-139.954,169.655,51.464,159.931
C04173=1016.647,290.548,-139.923,169.650,51.469,159.931
C04174=1016.641,290.301,-139.892,169.645,51.475,159.932
C04175=1016.636,290.053,-139.862,169.639,51.480,159.932
C04176=1016.629,289.804,-139.831,169.633,51.486,159.932
C04177=1016.623,289.557,-139.800,169.628,51.491,159.932
C04178=1016.617,289.309,-139.769,169.622,51.496,159.932
C04179=1016.612,289.060,-139.738,169.617,51.501,159.933
C04180=1016.606,288.813,-139.708,169.611,51.508,159.933
C04181=1016.599,288.564,-139.677,169.606,51.513,159.933
C04182=1016.593,288.316,-139.647,169.600,51.518,159.933
C04183=1016.587,288.068,-139.616,169.595,51.524,159.934
C04184=1016.581,287.821,-139.585,169.589,51.529,159.934
C04185=1016.575,287.573,-139.555,169.584,51.534,159.934
C04186=1016.569,287.324,-139.524,169.579,51.540,159.934
C04187=1016.563,287.076,-139.494,169.573,51.545,159.934
C04188=1016.557,286.829,-139.464,169.567,51.552,159.935
C04189=1016.551,286.580,-139.433,169.562,51.557,159.935
C04190=1016.545,286.332,-139.402,169.557,51.563,159.935
C04191=1016.539,286.084,-139.372,169.552,51.568,159.936
C04192=1016.533,285.837,-139.342,169.546,51.574,159.936
C04193=1016.527,285.588,-139.311,169.540,51.579,159.936
C04194=1016.521,285.340,-139.281,169.535,51.585,159.936
C04195=1016.515,285.092,-139.251,169.530,51.590,159.937
C04196=1016.509,284.843,-139.220,169.524,51.596,159.937
C04197=1016.503,284.595,-139.190,169.518,51.602,159.937
C04198=1016.497,284.348,-139.160,169.513,51.608,159.938
C04199=1016.491,284.100,-139.130,169.508,51.613,159.938
C04200=1016.485,283.852,-139.100,169.502,51.619,159.938
C04201=1016.479,283.603,-139.070,169.497,51.625,159.938
C04202=1016.472,283.356,-139.040,169.492,51.631,159.939
C04203=1016.467,283.107,-139.010,169.486,51.636,159.939
C04204=1016.461,282.859,-138.980,169.481,51.642,159.939
C04205=1016.455,282.611,-138.949,169.476,51.648,159.940
C04206=1016.448,282.363,-138.920,169.470,51.653,159.940
C04207=1016.443,282.115,-138.890,169.465,51.659,159.940
C04208=1016.437,281.867,-138.859,169.460,51.665,159.941
C04209=1016.431,281.619,-138.830,169.455,51.671,159.941
C04210=1016.425,281.371,-138.800,169.449,51.677,159.941
C04211=1016.419,281.122,-138.770,169.443,51.682,159.941
C04212=1016.413,280.874,-138.740,169.438,51.688,159.942
C04213=1016.406,280.626,-138.711,169.432,51.695,159.942
C04214=1016.401,280.378,-138.680,169.427,51.700,159.942
C04215=1016.395,280.130,-138.651,169.422,51.706,159.943
C04216=1016.389,279.882,-138.620,169.417,51.713,159.943
C04217=1016.383,279.634,-138.591,169.412,51.718,159.944
C04218=1016.377,279.386,-138.561,169.407,51.724,159.944
C04219=1016.371,279.168,-138.535,169.401,51.729,159.944
C04220=1016.367,278.951,-138.508,169.397,51.734,159.944
C04221=1016.362,278.734,-138.482,169.393,51.740,159.945
C04222=1016.356,278.517,-138.456,169.388,51.745,159.945
C04223=1016.351,278.300,-138.431,169.383,51.750,159.945
C04224=1016.347,278.083,-138.404,169.378,51.756,159.946
C04225=1016.341,277.866,-138.378,169.374,51.761,159.946
C04226=1016.332,277.478,-138.332,169.366,51.770,159.947
C04227=1016.326,277.230,-138.302,169.360,51.776,159.947
C04228=1016.321,276.982,-138.272,169.355,51.782,159.947
C04229=1016.315,276.733,-138.243,169.350,51.788,159.948
C04230=1016.309,276.486,-138.213,169.344,51.794,159.948
C04231=1016.303,276.237,-138.183,169.339,51.800,159.948
C04232=1016.298,275.989,-138.154,169.334,51.806,159.949
C04233=1016.291,275.741,-138.125,169.328,51.812,159.949
C04234=1016.285,275.493,-138.095,169.324,51.819,159.950
C04235=1016.279,275.245,-138.065,169.319,51.825,159.950
C04236=1016.273,274.996,-138.036,169.313,51.831,159.950
C04237=1016.268,274.748,-138.007,169.308,51.837,159.951
C04238=1016.261,274.500,-137.978,169.303,51.844,159.951
C04239=1016.256,274.251,-137.948,169.298,51.850,159.952
C04240=1016.250,274.003,-137.919,169.293,51.855,159.952
C04241=1016.244,273.755,-137.889,169.287,51.862,159.953
C04242=1016.238,273.507,-137.861,169.282,51.868,159.953
C04243=1016.233,273.259,-137.831,169.277,51.874,159.953
C04244=1016.227,273.011,-137.802,169.272,51.881,159.954
C04245=1016.221,272.762,-137.772,169.267,51.887,159.954
C04246=1016.215,272.514,-137.743,169.261,51.893,159.955
C04247=1016.209,272.266,-137.714,169.256,51.900,159.955
C04248=1016.203,272.018,-137.685,169.251,51.906,159.956
C04249=1016.197,271.770,-137.655,169.246,51.912,159.956
C04250=1016.192,271.522,-137.626,169.241,51.919,159.956
C04251=1016.186,271.274,-137.597,169.235,51.925,159.957
C04252=1016.180,271.025,-137.568,169.231,51.931,159.957
C04253=1016.174,270.777,-137.539,169.226,51.937,159.958
C04254=1016.168,270.528,-137.510,169.220,51.944,159.958
C04255=1016.162,270.280,-137.481,169.215,51.950,159.959
C04256=1016.157,270.033,-137.452,169.210,51.957,159.959
C04257=1016.151,269.784,-137.423,169.205,51.963,159.960
C04258=1016.145,269.535,-137.394,169.199,51.970,159.960
C04259=1016.139,269.287,-137.365,169.195,51.977,159.961
C04260=1016.134,269.039,-137.336,169.190,51.982,159.961
C04261=1016.128,268.791,-137.307,169.184,51.989,159.962
C04262=1016.122,268.543,-137.278,169.179,51.995,159.962
C04263=1016.116,268.294,-137.249,169.174,52.002,159.962
C04264=1016.111,268.047,-137.220,169.169,52.009,159.963
C04265=1016.105,267.798,-137.192,169.164,52.016,159.964
C04266=1016.099,267.550,-137.163,169.159,52.022,159.964
C04267=1016.093,267.301,-137.134,169.153,52.029,159.964
C04268=1016.087,267.054,-137.106,169.149,52.035,159.965
C04269=1016.082,266.805,-137.077,169.144,52.041,159.965
C04270=1016.076,266.556,-137.048,169.138,52.048,159.966
C04271=1016.070,266.308,-137.020,169.134,52.055,159.967
C04272=1016.064,266.060,-136.991,169.128,52.062,159.967
C04273=1016.058,265.812,-136.962,169.124,52.068,159.968
C04274=1016.053,265.564,-136.933,169.118,52.075,159.968
C04275=1016.047,265.315,-136.905,169.114,52.081,159.969
C04276=1016.041,265.067,-136.876,169.108,52.088,159.969
C04277=1016.036,264.819,-136.848,169.104,52.095,159.970
C04278=1016.029,264.571,-136.819,169.098,52.102,159.970
C04279=1016.025,264.334,-136.792,169.094,52.108,159.971
C04280=1016.018,264.098,-136.765,169.089,52.114,159.971
C04281=1016.013,263.862,-136.738,169.084,52.121,159.972
C04282=1016.008,263.625,-136.710,169.080,52.127,159.972
C04283=1016.002,263.389,-136.683,169.074,52.134,159.973
C04284=1015.997,263.153,-136.656,169.069,52.140,159.973
C04285=1015.991,262.916,-136.629,169.065,52.147,159.974
C04286=1015.986,262.680,-136.602,169.060,52.154,159.974
C04287=1015.980,262.432,-136.574,169.055,52.161,159.975
C04288=1015.974,262.184,-136.545,169.050,52.167,159.976
C04289=1015.968,261.935,-136.517,169.045,52.174,159.976
C04290=1015.963,261.687,-136.489,169.040,52.181,159.977
C04291=1015.957,261.439,-136.461,169.035,52.188,159.977
C04292=1015.951,261.191,-136.433,169.030,52.194,159.978
C04293=1015.945,260.942,-136.404,169.025,52.201,159.978
C04294=1015.941,260.694,-136.375,169.020,52.208,159.979
C04295=1015.935,260.445,-136.347,169.015,52.215,159.979
C04296=1015.929,260.197,-136.319,169.010,52.223,159.980
C04297=1015.923,259.949,-136.291,169.005,52.229,159.981
C04298=1015.918,259.701,-136.263,169.000,52.236,159.981
C04299=1015.911,259.452,-136.235,168.995,52.243,159.982
C04300=1015.906,259.204,-136.207,168.990,52.251,159.982
C04301=1015.900,258.955,-136.179,168.985,52.258,159.983
C04302=1015.894,258.708,-136.151,168.980,52.264,159.984
C04303=1015.888,258.459,-136.123,168.975,52.272,159.984
C04304=1015.882,258.211,-136.096,168.970,52.279,159.985
C04305=1015.876,257.962,-136.067,168.966,52.286,159.986
C04306=1015.871,257.714,-136.040,168.960,52.293,159.986
C04307=1015.864,257.465,-136.012,168.955,52.301,159.987
C04308=1015.859,257.217,-135.984,168.951,52.308,159.987
C04309=1015.853,256.969,-135.957,168.946,52.315,159.988
C04310=1015.847,256.720,-135.929,168.940,52.322,159.989
C04311=1015.842,256.472,-135.902,168.936,52.330,159.989
C04312=1015.835,256.224,-135.874,168.931,52.337,159.990
C04313=1015.830,255.975,-135.846,168.926,52.344,159.991
C04314=1015.824,255.726,-135.818,168.921,52.351,159.991
C04315=1015.818,255.478,-135.791,168.916,52.359,159.992
C04316=1015.813,255.230,-135.763,168.911,52.366,159.992
C04317=1015.806,254.981,-135.736,168.906,52.373,159.993
C04318=1015.801,254.733,-135.708,168.902,52.381,159.994
C04319=1015.795,254.484,-135.680,168.896,52.388,159.995
C04320=1015.789,254.236,-135.653,168.891,52.395,159.995
C04321=1015.784,253.988,-135.625,168.887,52.403,159.996
C04322=1015.777,253.740,-135.597,168.882,52.410,159.997
C04323=1015.772,253.491,-135.570,168.877,52.417,159.997
C04324=1015.767,253.243,-135.542,168.873,52.425,159.998
C04325=1015.761,252.994,-135.515,168.867,52.432,159.999
C04326=1015.755,252.746,-135.487,168.862,52.440,159.999
C04327=1015.750,252.498,-135.459,168.857,52.447,160.000
C04328=1015.743,252.249,-135.432,168.853,52.454,160.001
C04329=1015.738,252.001,-135.404,168.848,52.462,160.001
C04330=1015.732,251.752,-135.377,168.843,52.469,160.002
C04331=1015.727,251.504,-135.350,168.838,52.477,160.003
C04332=1015.721,251.255,-135.322,168.833,52.484,160.003
C04333=1015.715,251.007,-135.295,168.828,52.491,160.004
C04334=1015.710,250.758,-135.267,168.823,52.499,160.005
C04335=1015.704,250.510,-135.240,168.819,52.507,160.006
C04336=1015.699,250.261,-135.212,168.814,52.514,160.006
C04337=1015.693,250.013,-135.185,168.809,52.522,160.007
C04338=1015.687,249.765,-135.158,168.804,52.529,160.008
C04339=1015.682,249.527,-135.132,168.800,52.536,160.008
C04340=1015.677,249.291,-135.106,168.796,52.544,160.009
C04341=1015.672,249.053,-135.079,168.791,52.551,160.010
C04342=1015.666,248.816,-135.053,168.787,52.558,160.010
C04343=1015.661,248.578,-135.027,168.781,52.565,160.011
C04344=1015.655,248.341,-135.001,168.777,52.573,160.012
C04345=1015.651,248.104,-134.975,168.772,52.580,160.012
C04346=1015.645,247.867,-134.949,168.768,52.587,160.013
C04347=1015.640,247.619,-134.921,168.763,52.595,160.014
C04348=1015.634,247.370,-134.895,168.759,52.602,160.015
C04349=1015.629,247.122,-134.867,168.754,52.610,160.015
C04350=1015.623,246.873,-134.839,168.749,52.618,160.016
C04351=1015.618,246.625,-134.813,168.744,52.625,160.017
C04352=1015.613,246.376,-134.786,168.739,52.633,160.017
C04353=1015.606,246.128,-134.758,168.735,52.640,160.018
C04354=1015.601,245.879,-134.731,168.730,52.648,160.019
C04355=1015.596,245.631,-134.703,168.725,52.656,160.020
C04356=1015.590,245.382,-134.677,168.720,52.664,160.020
C04357=1015.585,245.134,-134.649,168.715,52.671,160.021
C04358=1015.579,244.886,-134.622,168.711,52.679,160.022
C04359=1015.574,244.637,-134.595,168.706,52.687,160.023
C04360=1015.568,244.389,-134.568,168.701,52.695,160.024
C04361=1015.563,244.140,-134.541,168.696,52.703,160.024
C04362=1015.558,243.891,-134.514,168.691,52.711,160.025
C04363=1015.552,243.644,-134.486,168.687,52.718,160.026
C04364=1015.547,243.395,-134.459,168.682,52.726,160.027
C04365=1015.541,243.147,-134.432,168.678,52.734,160.027
C04366=1015.536,242.898,-134.405,168.673,52.742,160.028
C04367=1015.530,242.650,-134.379,168.668,52.750,160.029
C04368=1015.525,242.401,-134.351,168.663,52.757,160.030
C04369=1015.520,242.153,-134.325,168.659,52.766,160.031
C04370=1015.514,241.904,-134.298,168.654,52.773,160.031
C04371=1015.509,241.656,-134.271,168.650,52.781,160.032
C04372=1015.503,241.407,-134.244,168.645,52.790,160.033
C04373=1015.497,241.159,-134.218,168.640,52.797,160.034
C04374=1015.492,240.910,-134.192,168.636,52.806,160.035
C04375=1015.487,240.661,-134.164,168.631,52.814,160.035
C04376=1015.481,240.413,-134.138,168.626,52.822,160.036
C04377=1015.475,240.165,-134.111,168.621,52.830,160.037
C04378=1015.470,239.916,-134.084,168.617,52.838,160.038
C04379=1015.464,239.667,-134.057,168.612,52.846,160.039
C04380=1015.459,239.419,-134.031,168.607,52.854,160.039
C04381=1015.454,239.170,-134.004,168.602,52.862,160.040
C04382=1015.448,238.921,-133.977,168.598,52.871,160.041
C04383=1015.442,238.673,-133.951,168.593,52.879,160.042
C04384=1015.437,238.425,-133.925,168.588,52.887,160.043
C04385=1015.432,238.176,-133.898,168.583,52.895,160.044
C04386=1015.426,237.928,-133.872,168.579,52.903,160.045
C04387=1015.420,237.679,-133.846,168.574,52.912,160.045
C04388=1015.415,237.431,-133.819,168.569,52.920,160.046
C04389=1015.409,237.182,-133.793,168.565,52.928,160.047
C04390=1015.403,236.933,-133.767,168.560,52.937,160.048
C04391=1015.398,236.685,-133.740,168.556,52.945,160.049
C04392=1015.393,236.437,-133.714,168.551,52.953,160.050
C04393=1015.387,236.188,-133.688,168.546,52.961,160.051
C04394=1015.382,235.939,-133.662,168.542,52.970,160.052
C04395=1015.376,235.691,-133.635,168.537,52.978,160.053
C04396=1015.370,235.442,-133.609,168.533,52.987,160.053
C04397=1015.365,235.194,-133.583,168.528,52.995,160.054
C04398=1015.359,234.945,-133.557,168.523,53.003,160.055
C04399=1015.354,234.705,-133.532,168.519,53.012,160.056
C04400=1015.348,234.464,-133.506,168.515,53.020,160.057
C04401=1015.344,234.223,-133.480,168.510,53.028,160.058
C04402=1015.339,233.983,-133.455,168.505,53.036,160.059
C04403=1015.333,233.742,-133.430,168.501,53.045,160.060
C04404=1015.328,233.501,-133.404,168.496,53.053,160.060
C04405=1015.323,233.262,-133.379,168.492,53.061,160.061
C04406=1015.317,233.020,-133.354,168.488,53.069,160.062
C04407=1015.311,232.772,-133.328,168.483,53.078,160.063
C04408=1015.306,232.523,-133.302,168.478,53.087,160.064
C04409=1015.301,232.275,-133.276,168.473,53.095,160.065
C04410=1015.295,232.026,-133.250,168.469,53.104,160.066
C04411=1015.290,231.777,-133.224,168.464,53.112,160.067
C04412=1015.284,231.528,-133.198,168.460,53.121,160.068
C04413=1015.278,231.281,-133.172,168.455,53.129,160.069
C04414=1015.273,231.032,-133.146,168.451,53.138,160.070
C04415=1015.268,230.783,-133.120,168.446,53.147,160.070
C04416=1015.263,230.535,-133.095,168.441,53.155,160.071
C04417=1015.257,230.286,-133.068,168.437,53.164,160.072
C04418=1015.251,230.037,-133.042,168.432,53.172,160.073
C04419=1015.247,229.789,-133.017,168.428,53.181,160.074
C04420=1015.241,229.540,-132.991,168.422,53.190,160.075
C04421=1015.236,229.291,-132.965,168.418,53.199,160.076
C04422=1015.230,229.044,-132.938,168.414,53.208,160.077
C04423=1015.224,228.795,-132.913,168.409,53.216,160.078
C04424=1015.219,228.546,-132.887,168.405,53.225,160.079
C04425=1015.214,228.298,-132.862,168.400,53.234,160.080
C04426=1015.208,228.049,-132.836,168.396,53.243,160.081
C04427=1015.203,227.800,-132.810,168.391,53.251,160.082
C04428=1015.197,227.552,-132.785,168.386,53.261,160.083
C04429=1015.192,227.303,-132.759,168.382,53.270,160.084
C04430=1015.186,227.054,-132.733,168.377,53.278,160.085
C04431=1015.182,226.805,-132.707,168.373,53.287,160.086
C04432=1015.176,226.556,-132.681,168.368,53.296,160.087
C04433=1015.171,226.309,-132.656,168.363,53.305,160.088
C04434=1015.165,226.060,-132.630,168.359,53.314,160.089
C04435=1015.160,225.811,-132.604,168.354,53.323,160.090
C04436=1015.154,225.563,-132.580,168.350,53.332,160.091
C04437=1015.149,225.314,-132.554,168.346,53.341,160.092
C04438=1015.143,225.065,-132.529,168.341,53.351,160.093
C04439=1015.138,224.816,-132.503,168.336,53.359,160.094
C04440=1015.132,224.567,-132.478,168.331,53.369,160.095
C04441=1015.127,224.319,-132.453,168.327,53.378,160.096
C04442=1015.120,224.070,-132.427,168.323,53.387,160.097
C04443=1015.116,223.822,-132.402,168.318,53.396,160.098
C04444=1015.110,223.573,-132.376,168.313,53.405,160.099
C04445=1015.105,223.325,-132.351,168.309,53.415,160.100
C04446=1015.099,223.076,-132.325,168.305,53.424,160.101
C04447=1015.094,222.827,-132.301,168.300,53.432,160.102
C04448=1015.089,222.578,-132.275,168.295,53.442,160.103
C04449=1015.083,222.330,-132.250,168.291,53.451,160.104
C04450=1015.078,222.080,-132.225,168.286,53.460,160.105
C04451=1015.072,221.832,-132.200,168.282,53.470,160.106
C04452=1015.067,221.584,-132.174,168.277,53.479,160.107
C04453=1015.061,221.335,-132.150,168.273,53.488,160.109
C04454=1015.056,221.086,-132.124,168.268,53.497,160.109
C04455=1015.050,220.838,-132.099,168.264,53.507,160.111
C04456=1015.045,220.588,-132.074,168.260,53.516,160.112
C04457=1015.040,220.340,-132.048,168.255,53.526,160.113
C04458=1015.034,220.091,-132.023,168.250,53.534,160.114
C04459=1015.029,219.847,-131.999,168.246,53.544,160.115
C04460=1015.024,219.602,-131.974,168.242,53.553,160.116
C04461=1015.018,219.357,-131.949,168.238,53.563,160.117
C04462=1015.013,219.113,-131.924,168.232,53.572,160.118
C04463=1015.008,218.867,-131.899,168.228,53.581,160.119
C04464=1015.003,218.623,-131.875,168.223,53.591,160.120
C04465=1014.998,218.379,-131.850,168.219,53.599,160.121
C04466=1014.992,218.134,-131.825,168.215,53.608,160.122
C04467=1014.987,217.885,-131.801,168.210,53.618,160.123
C04468=1014.982,217.636,-131.775,168.206,53.627,160.125
C04469=1014.976,217.388,-131.751,168.201,53.637,160.126
C04470=1014.971,217.139,-131.726,168.197,53.647,160.127
C04471=1014.965,216.890,-131.701,168.193,53.656,160.128
C04472=1014.960,216.641,-131.676,168.188,53.667,160.129
C04473=1014.955,216.393,-131.652,168.183,53.676,160.130
C04474=1014.949,216.144,-131.627,168.179,53.686,160.131
C04475=1014.943,215.896,-131.602,168.175,53.695,160.132
C04476=1014.939,215.647,-131.577,168.170,53.705,160.134
C04477=1014.933,215.398,-131.552,168.166,53.714,160.135
C04478=1014.927,215.149,-131.528,168.161,53.725,160.136
C04479=1014.922,214.901,-131.504,168.156,53.734,160.137
C04480=1014.916,214.652,-131.479,168.153,53.744,160.138
C04481=1014.911,214.403,-131.453,168.148,53.754,160.139
C04482=1014.906,214.155,-131.429,168.143,53.764,160.141
C04483=1014.900,213.905,-131.404,168.139,53.773,160.142
C04484=1014.895,213.657,-131.380,168.135,53.783,160.143
C04485=1014.890,213.408,-131.355,168.130,53.793,160.144
C04486=1014.885,213.160,-131.330,168.125,53.803,160.145
C04487=1014.879,212.911,-131.306,168.121,53.812,160.146
C04488=1014.873,212.662,-131.282,168.116,53.822,160.147
C04489=1014.869,212.413,-131.257,168.112,53.833,160.149
C04490=1014.864,212.165,-131.232,168.108,53.842,160.150
C04491=1014.858,211.915,-131.208,168.103,53.852,160.151
C04492=1014.852,211.667,-131.184,168.099,53.862,160.152
C04493=1014.847,211.419,-131.159,168.094,53.872,160.153
C04494=1014.842,211.170,-131.134,168.091,53.882,160.155
C04495=1014.836,210.921,-131.109,168.086,53.892,160.156
C04496=1014.831,210.672,-131.085,168.081,53.901,160.157
C04497=1014.826,210.423,-131.061,168.077,53.912,160.158
C04498=1014.821,210.174,-131.036,168.072,53.922,160.159
C04499=1014.816,209.926,-131.011,168.068,53.932,160.161
C04500=1014.810,209.677,-130.987,168.064,53.941,160.162
C04501=1014.805,209.428,-130.963,168.059,53.952,160.163
C04502=1014.799,209.179,-130.938,168.054,53.962,160.164
C04503=1014.794,208.931,-130.914,168.050,53.972,160.165
C04504=1014.789,208.682,-130.890,168.046,53.983,160.167
C04505=1014.783,208.434,-130.866,168.042,53.992,160.168
C04506=1014.778,208.184,-130.841,168.037,54.002,160.169
C04507=1014.772,207.936,-130.817,168.033,54.013,160.170
C04508=1014.767,207.687,-130.792,168.028,54.023,160.171
C04509=1014.762,207.438,-130.769,168.024,54.033,160.173
C04510=1014.757,207.189,-130.744,168.020,54.044,160.174
C04511=1014.752,206.940,-130.720,168.015,54.053,160.175
C04512=1014.746,206.692,-130.696,168.010,54.064,160.176
C04513=1014.741,206.444,-130.672,168.006,54.074,160.178
C04514=1014.736,206.195,-130.648,168.002,54.085,160.179
C04515=1014.731,205.946,-130.624,167.997,54.095,160.180
C04516=1014.725,205.697,-130.599,167.993,54.105,160.181
C04517=1014.719,205.448,-130.575,167.988,54.116,160.183
C04518=1014.714,205.199,-130.551,167.984,54.126,160.184
C04519=1014.709,204.968,-130.529,167.980,54.136,160.185
C04520=1014.705,204.736,-130.506,167.976,54.145,160.186
C04521=1014.699,204.503,-130.484,167.972,54.155,160.188
C04522=1014.694,204.272,-130.462,167.968,54.165,160.189
C04523=1014.689,204.039,-130.440,167.963,54.175,160.190
C04524=1014.685,203.808,-130.418,167.960,54.185,160.191
C04525=1014.680,203.576,-130.395,167.955,54.195,160.192
C04526=1014.674,203.344,-130.373,167.952,54.204,160.194
C04527=1014.655,202.228,-130.273,167.429,54.129,160.062
C04528=1014.651,201.979,-130.251,167.424,54.141,160.063
C04529=1014.646,201.730,-130.229,167.419,54.153,160.064
C04530=1014.642,201.481,-130.207,167.415,54.164,160.066
C04531=1014.638,201.232,-130.185,167.410,54.176,160.067
C04532=1014.634,200.983,-130.163,167.405,54.187,160.069
C04533=1014.630,200.734,-130.140,167.400,54.199,160.070
C04534=1014.625,200.485,-130.118,167.396,54.210,160.071
C04535=1014.621,200.236,-130.096,167.391,54.222,160.073
C04536=1014.617,199.987,-130.073,167.386,54.233,160.074
C04537=1014.612,199.738,-130.052,167.382,54.245,160.075
C04538=1014.608,199.489,-130.030,167.378,54.256,160.077
C04539=1014.605,199.240,-130.008,167.373,54.268,160.078
C04540=1014.600,198.991,-129.986,167.368,54.280,160.079
C04541=1014.596,198.742,-129.963,167.363,54.291,160.081
C04542=1014.591,198.494,-129.941,167.359,54.303,160.082
C04543=1014.587,198.244,-129.920,167.354,54.314,160.084
C04544=1014.583,197.995,-129.898,167.349,54.326,160.085
C04545=1014.578,197.745,-129.877,167.344,54.338,160.086
C04546=1014.574,197.497,-129.855,167.339,54.349,160.087
C04547=1014.570,197.248,-129.833,167.335,54.361,160.089
C04548=1014.565,196.999,-129.812,167.331,54.372,160.090
C04549=1014.560,196.750,-129.790,167.326,54.384,160.092
C04550=1014.556,196.501,-129.769,167.321,54.396,160.093
C04551=1014.552,196.252,-129.747,167.316,54.408,160.094
C04552=1014.548,196.003,-129.725,167.312,54.419,160.096
C04553=1014.543,195.754,-129.704,167.308,54.431,160.097
C04554=1014.539,195.505,-129.681,167.303,54.443,160.099
C04555=1014.535,195.256,-129.660,167.298,54.454,160.100
C04556=1014.530,195.007,-129.638,167.294,54.466,160.101
C04557=1014.526,194.758,-129.617,167.289,54.477,160.103
C04558=1014.522,194.509,-129.595,167.284,54.489,160.104
C04559=1014.518,194.260,-129.574,167.279,54.501,160.105
C04560=1014.513,194.011,-129.552,167.275,54.512,160.107
C04561=1014.508,193.762,-129.531,167.271,54.524,160.108
C04562=1014.505,193.512,-129.509,167.266,54.536,160.109
C04563=1014.500,193.264,-129.488,167.262,54.548,160.111
C04564=1014.496,193.014,-129.467,167.258,54.559,160.112
C04565=1014.492,192.765,-129.444,167.253,54.571,160.114
C04566=1014.488,192.517,-129.423,167.249,54.582,160.115
C04567=1014.483,192.268,-129.402,167.244,54.594,160.117
C04568=1014.478,192.018,-129.380,167.239,54.606,160.118
C04569=1014.475,191.769,-129.359,167.235,54.617,160.119
C04570=1014.470,191.520,-129.337,167.231,54.629,160.121
C04571=1014.466,191.271,-129.316,167.226,54.641,160.122
C04572=1014.462,191.022,-129.295,167.222,54.652,160.124
C04573=1014.458,190.773,-129.273,167.217,54.664,160.125
C04574=1014.454,190.524,-129.252,167.212,54.676,160.126
C04575=1014.450,190.275,-129.231,167.208,54.687,160.128
C04576=1014.445,190.026,-129.208,167.204,54.699,160.129
C04577=1014.442,189.777,-129.188,167.199,54.710,160.130
C04578=1014.437,189.528,-129.166,167.195,54.722,160.132
C04579=1014.433,189.280,-129.145,167.190,54.734,160.133
C04580=1014.429,189.030,-129.123,167.186,54.745,160.135
C04581=1014.424,188.780,-129.102,167.182,54.757,160.136
C04582=1014.420,188.532,-129.081,167.178,54.768,160.137
C04583=1014.416,188.283,-129.059,167.173,54.780,160.139
C04584=1014.413,188.034,-129.038,167.168,54.792,160.140
C04585=1014.408,187.784,-129.017,167.164,54.803,160.141
C04586=1014.404,187.536,-128.996,167.160,54.815,160.143
C04587=1014.400,187.286,-128.974,167.156,54.826,160.144
C04588=1014.396,187.007,-128.950,167.151,54.840,160.146
C04589=1014.391,186.727,-128.926,167.146,54.853,160.147
C04590=1014.386,186.448,-128.902,167.142,54.865,160.149
C04591=1014.382,186.169,-128.879,167.137,54.879,160.151
C04592=1014.377,185.920,-128.857,167.133,54.890,160.152
C04593=1014.373,185.671,-128.836,167.128,54.902,160.154
C04594=1014.369,185.422,-128.815,167.125,54.913,160.155
C04595=1014.366,185.173,-128.794,167.120,54.925,160.156
C04596=1014.361,184.923,-128.773,167.116,54.937,160.158
C04597=1014.357,184.675,-128.752,167.111,54.948,160.159
C04598=1014.353,184.425,-128.731,167.108,54.960,160.161
C04599=1014.350,184.176,-128.709,167.103,54.972,160.162
C04600=1014.345,183.927,-128.687,167.099,54.983,160.163
C04601=1014.341,183.679,-128.667,167.094,54.995,160.165
C04602=1014.336,183.429,-128.645,167.090,55.006,160.166
C04603=1014.333,183.180,-128.624,167.085,55.018,160.167
C04604=1014.329,182.931,-128.603,167.082,55.029,160.169
C04605=1014.325,182.682,-128.582,167.078,55.040,160.170
C04606=1014.321,182.433,-128.561,167.073,55.052,160.172
C04607=1014.317,182.183,-128.540,167.070,55.064,160.173
C04608=1014.313,181.935,-128.519,167.065,55.075,160.174
C04609=1014.309,181.685,-128.498,167.061,55.087,160.176
C04610=1014.305,181.437,-128.477,167.057,55.098,160.177
C04611=1014.300,181.186,-128.456,167.053,55.110,160.179
C04612=1014.296,180.938,-128.436,167.049,55.123,160.180
C04613=1014.292,180.689,-128.415,167.045,55.134,160.182
C04614=1014.288,180.439,-128.395,167.040,55.146,160.183
C04615=1014.283,180.191,-128.375,167.037,55.158,160.185
C04616=1014.279,179.941,-128.354,167.032,55.170,160.186
C04617=1014.275,179.692,-128.334,167.028,55.182,160.188
C04618=1014.270,179.444,-128.313,167.024,55.193,160.189
C04619=1014.266,179.194,-128.293,167.019,55.205,160.190
C04620=1014.261,178.945,-128.273,167.016,55.217,160.192
C04621=1014.257,178.695,-128.252,167.011,55.229,160.194
C04622=1014.253,178.446,-128.232,167.008,55.241,160.195
C04623=1014.249,178.198,-128.211,167.003,55.253,160.196
C04624=1014.244,177.948,-128.191,167.000,55.264,160.198
C04625=1014.240,177.699,-128.171,166.995,55.276,160.199
C04626=1014.236,177.450,-128.151,166.992,55.288,160.201
C04627=1014.232,177.201,-128.130,166.987,55.300,160.202
C04628=1014.227,176.952,-128.110,166.983,55.312,160.204
C04629=1014.223,176.703,-128.089,166.979,55.324,160.205
C04630=1014.218,176.453,-128.070,166.975,55.335,160.207
C04631=1014.214,176.204,-128.049,166.971,55.348,160.208
C04632=1014.211,175.955,-128.029,166.967,55.359,160.210
C04633=1014.206,175.706,-128.008,166.963,55.371,160.211
C04634=1014.202,175.457,-127.988,166.959,55.383,160.213
C04635=1014.197,175.208,-127.968,166.955,55.394,160.214
C04636=1014.194,174.959,-127.948,166.951,55.406,160.215
C04637=1014.189,174.709,-127.927,166.946,55.418,160.217
C04638=1014.185,174.460,-127.907,166.943,55.430,160.218
C04639=1014.181,174.211,-127.887,166.939,55.442,160.220
C04640=1014.177,173.963,-127.867,166.935,55.453,160.221
C04641=1014.172,173.713,-127.846,166.931,55.465,160.223
C04642=1014.168,173.464,-127.826,166.927,55.477,160.224
C04643=1014.164,173.215,-127.806,166.923,55.488,160.226
C04644=1014.160,172.965,-127.786,166.919,55.500,160.227
C04645=1014.155,172.716,-127.766,166.915,55.512,160.229
C04646=1014.152,172.467,-127.746,166.912,55.524,160.230
C04647=1014.148,172.218,-127.725,166.907,55.536,160.232
C04648=1014.143,171.969,-127.705,166.904,55.548,160.233
C04649=1014.140,171.720,-127.685,166.900,55.559,160.235
C04650=1014.134,171.471,-127.665,166.896,55.571,160.236
C04651=1014.131,171.221,-127.645,166.892,55.583,160.238
C04652=1014.126,170.942,-127.622,166.887,55.596,160.239
C04653=1014.121,170.662,-127.600,166.884,55.609,160.241
C04654=1014.117,170.382,-127.577,166.879,55.622,160.242
C04655=1014.113,170.103,-127.555,166.875,55.636,160.244
C04656=1014.109,169.854,-127.534,166.871,55.647,160.246
C04657=1014.104,169.605,-127.515,166.867,55.659,160.247
C04658=1014.101,169.356,-127.495,166.863,55.671,160.249
C04659=1014.096,169.107,-127.474,166.860,55.682,160.250
C04660=1014.092,168.858,-127.454,166.855,55.694,160.251
C04661=1014.087,168.608,-127.434,166.852,55.706,160.253
C04662=1014.084,168.359,-127.414,166.848,55.717,160.254
C04663=1014.080,168.109,-127.394,166.845,55.729,160.256
C04664=1014.076,167.861,-127.374,166.840,55.741,160.257
C04665=1014.072,167.612,-127.354,166.837,55.752,160.259
C04666=1014.068,167.363,-127.335,166.833,55.764,160.260
C04667=1014.064,167.113,-127.315,166.830,55.776,160.262
C04668=1014.060,166.864,-127.294,166.825,55.788,160.263
C04669=1014.056,166.616,-127.274,166.822,55.799,160.265
C04670=1014.052,166.366,-127.254,166.818,55.811,160.266
C04671=1014.047,166.116,-127.234,166.815,55.822,160.268
C04672=1014.044,165.867,-127.214,166.811,55.834,160.269
C04673=1014.039,165.618,-127.195,166.807,55.846,160.271
C04674=1014.036,165.369,-127.175,166.803,55.858,160.272
C04675=1014.032,165.120,-127.154,166.800,55.869,160.274
C04676=1014.027,164.871,-127.134,166.796,55.881,160.275
C04677=1014.024,164.622,-127.114,166.793,55.892,160.277
C04678=1014.019,164.372,-127.095,166.788,55.904,160.278
C04679=1014.016,164.123,-127.075,166.785,55.916,160.280
C04680=1014.011,163.874,-127.055,166.782,55.928,160.281
C04681=1014.008,163.625,-127.035,166.778,55.938,160.282
C04682=1014.004,163.375,-127.015,166.774,55.950,160.284
C04683=1014.000,163.126,-126.996,166.771,55.962,160.285
C04684=1013.996,162.877,-126.976,166.767,55.973,160.287
C04685=1013.992,162.629,-126.956,166.764,55.985,160.288
C04686=1013.988,162.379,-126.935,166.759,55.997,160.290
C04687=1013.984,162.130,-126.915,166.756,56.009,160.291
C04688=1013.980,161.881,-126.896,166.752,56.020,160.293
C04689=1013.976,161.631,-126.876,166.749,56.032,160.294
C04690=1013.972,161.382,-126.856,166.746,56.043,160.296
C04691=1013.968,161.133,-126.836,166.742,56.054,160.297
C04692=1013.964,160.884,-126.817,166.738,56.066,160.299
C04693=1013.960,160.635,-126.797,166.735,56.078,160.300
C04694=1013.957,160.385,-126.777,166.731,56.089,160.302
C04695=1013.953,160.136,-126.757,166.728,56.101,160.303
C04696=1013.950,159.888,-126.738,166.725,56.113,160.305
C04697=1013.945,159.639,-126.718,166.721,56.124,160.306
C04698=1013.942,159.389,-126.698,166.717,56.135,160.308
C04699=1013.937,159.140,-126.679,166.714,56.147,160.309
C04700=1013.934,158.890,-126.659,166.711,56.158,160.311
C04701=1013.930,158.641,-126.639,166.707,56.170,160.312
C04702=1013.926,158.392,-126.620,166.703,56.181,160.314
C04703=1013.922,158.142,-126.600,166.700,56.193,160.315
C04704=1013.918,157.893,-126.580,166.696,56.204,160.317
C04705=1013.914,157.644,-126.561,166.692,56.216,160.318
C04706=1013.910,157.395,-126.542,166.689,56.228,160.319
C04707=1013.905,157.146,-126.522,166.685,56.240,160.321
C04708=1013.901,156.896,-126.504,166.682,56.252,160.323
C04709=1013.897,156.647,-126.484,166.679,56.263,160.324
C04710=1013.893,156.398,-126.465,166.675,56.275,160.326
C04711=1013.889,156.148,-126.445,166.672,56.287,160.327
C04712=1013.885,155.900,-126.426,166.669,56.298,160.329
C04713=1013.881,155.650,-126.408,166.664,56.310,160.330
C04714=1013.877,155.401,-126.388,166.661,56.322,160.332
C04715=1013.873,155.152,-126.369,166.657,56.334,160.333
C04716=1013.868,154.872,-126.347,166.654,56.347,160.335
C04717=1013.863,154.592,-126.326,166.650,56.360,160.337
C04718=1013.859,154.312,-126.305,166.647,56.373,160.338
C04719=1013.855,154.032,-126.283,166.643,56.386,160.340
C04720=1013.850,153.783,-126.264,166.639,56.397,160.342
C04721=1013.846,153.534,-126.244,166.635,56.410,160.343
C04722=1013.842,153.284,-126.226,166.632,56.421,160.345
C04723=1013.838,153.036,-126.206,166.628,56.433,160.346
C04724=1013.834,152.786,-126.188,166.625,56.445,160.348
C04725=1013.831,152.537,-126.168,166.622,56.456,160.349
C04726=1013.827,152.287,-126.149,166.619,56.468,160.351
C04727=1013.823,152.038,-126.130,166.615,56.480,160.352
C04728=1013.817,151.789,-126.111,166.611,56.491,160.354
C04729=1013.814,151.540,-126.093,166.608,56.503,160.355
C04730=1013.810,151.291,-126.073,166.605,56.514,160.357
C04731=1013.806,151.041,-126.055,166.602,56.526,160.358
C04732=1013.801,150.792,-126.035,166.598,56.538,160.360
C04733=1013.798,150.543,-126.017,166.595,56.549,160.361
C04734=1013.794,150.294,-125.998,166.592,56.561,160.363
C04735=1013.789,150.045,-125.979,166.589,56.573,160.365
C04736=1013.785,149.795,-125.960,166.585,56.585,160.366
C04737=1013.781,149.545,-125.941,166.582,56.596,160.368
C04738=1013.778,149.297,-125.922,166.578,56.607,160.369
C04739=1013.774,149.047,-125.903,166.575,56.619,160.370
C04740=1013.770,148.798,-125.884,166.572,56.631,160.372
C04741=1013.765,148.549,-125.865,166.568,56.643,160.374
C04742=1013.762,148.300,-125.847,166.565,56.654,160.375
C04743=1013.758,148.050,-125.828,166.563,56.666,160.377
C04744=1013.753,147.801,-125.809,166.559,56.677,160.378
C04745=1013.749,147.552,-125.791,166.556,56.688,160.380
C04746=1013.745,147.303,-125.772,166.553,56.700,160.381
C04747=1013.741,147.053,-125.753,166.550,56.712,160.383
C04748=1013.737,146.804,-125.734,166.546,56.724,160.384
C04749=1013.733,146.555,-125.715,166.543,56.736,160.386
C04750=1013.729,146.305,-125.696,166.539,56.747,160.387
C04751=1013.724,146.056,-125.678,166.536,56.758,160.389
C04752=1013.721,145.808,-125.659,166.533,56.770,160.390
C04753=1013.717,145.558,-125.640,166.530,56.782,160.392
C04754=1013.713,145.308,-125.622,166.526,56.794,160.394
C04755=1013.709,145.059,-125.603,166.524,56.804,160.395
C04756=1013.704,144.810,-125.585,166.521,56.816,160.397
C04757=1013.700,144.560,-125.566,166.517,56.828,160.398
C04758=1013.697,144.311,-125.548,166.514,56.840,160.400
C04759=1013.692,144.062,-125.530,166.511,56.851,160.401
C04760=1013.688,143.812,-125.511,166.508,56.863,160.403
C04761=1013.685,143.563,-125.493,166.504,56.874,160.404
C04762=1013.680,143.314,-125.474,166.501,56.886,160.406
C04763=1013.676,143.065,-125.455,166.498,56.898,160.407
C04764=1013.672,142.816,-125.437,166.495,56.910,160.409
C04765=1013.667,142.567,-125.418,166.491,56.921,160.411
C04766=1013.663,142.317,-125.400,166.489,56.932,160.412
C04767=1013.660,142.068,-125.381,166.486,56.944,160.414
C04768=1013.655,141.819,-125.363,166.482,56.956,160.415
C04769=1013.651,141.569,-125.344,166.479,56.968,160.417
C04770=1013.648,141.320,-125.326,166.476,56.979,160.418
C04771=1013.643,141.071,-125.308,166.472,56.990,160.420
C04772=1013.639,140.822,-125.289,166.469,57.002,160.421
C04773=1013.635,140.572,-125.271,166.467,57.014,160.423
C04774=1013.631,140.323,-125.252,166.463,57.025,160.424
C04775=1013.627,140.073,-125.235,166.460,57.037,160.426
C04776=1013.623,139.824,-125.217,166.457,57.048,160.427
C04777=1013.619,139.575,-125.198,166.454,57.060,160.429
C04778=1013.615,139.325,-125.180,166.451,57.071,160.431
C04779=1013.611,139.077,-125.162,166.448,57.083,160.432
C04780=1013.606,138.796,-125.140,166.445,57.096,160.434
C04781=1013.602,138.517,-125.120,166.441,57.109,160.436
C04782=1013.597,138.237,-125.099,166.438,57.122,160.437
C04783=1013.593,137.957,-125.079,166.435,57.134,160.439
C04784=1013.589,137.707,-125.061,166.431,57.145,160.440
C04785=1013.585,137.458,-125.042,166.428,57.157,160.442
C04786=1013.580,137.209,-125.024,166.425,57.169,160.444
C04787=1013.577,136.960,-125.006,166.423,57.180,160.445
C04788=1013.573,136.710,-124.988,166.419,57.192,160.447
C04789=1013.569,136.461,-124.970,166.416,57.203,160.448
C04790=1013.564,136.212,-124.952,166.413,57.215,160.450
C04791=1013.560,135.963,-124.934,166.411,57.226,160.451
C04792=1013.556,135.713,-124.915,166.408,57.238,160.453
C04793=1013.552,135.464,-124.898,166.404,57.249,160.454
C04794=1013.548,135.215,-124.879,166.401,57.261,160.456
C04795=1013.544,134.966,-124.861,166.399,57.272,160.458
C04796=1013.540,134.716,-124.843,166.395,57.283,160.459
C04797=1013.536,134.467,-124.826,166.392,57.295,160.461
C04798=1013.532,134.217,-124.807,166.390,57.307,160.462
C04799=1013.528,133.968,-124.790,166.387,57.318,160.464
C04800=1013.523,133.719,-124.772,166.384,57.330,160.465
C04801=1013.520,133.470,-124.753,166.380,57.341,160.467
C04802=1013.515,133.220,-124.736,166.378,57.352,160.468
C04803=1013.511,132.971,-124.718,166.375,57.364,160.470
C04804=1013.507,132.721,-124.699,166.371,57.375,160.471
C04805=1013.503,132.472,-124.682,166.369,57.387,160.473
C04806=1013.499,132.222,-124.663,166.366,57.398,160.474
C04807=1013.495,131.973,-124.646,166.363,57.410,160.476
C04808=1013.491,131.724,-124.628,166.360,57.421,160.478
C04809=1013.487,131.475,-124.610,166.357,57.432,160.479
C04810=1013.483,131.225,-124.592,166.355,57.443,160.481
C04811=1013.479,130.976,-124.575,166.352,57.455,160.482
C04812=1013.475,130.727,-124.557,166.348,57.466,160.484
C04813=1013.471,130.477,-124.539,166.346,57.478,160.485
C04814=1013.467,130.228,-124.520,166.343,57.489,160.487
C04815=1013.463,129.978,-124.503,166.341,57.500,160.489
C04816=1013.459,129.730,-124.485,166.337,57.512,160.490
C04817=1013.455,129.479,-124.467,166.334,57.523,160.491
C04818=1013.451,129.231,-124.449,166.332,57.534,160.493
C04819=1013.446,128.981,-124.432,166.329,57.546,160.495
C04820=1013.442,128.732,-124.415,166.325,57.557,160.496
C04821=1013.438,128.483,-124.397,166.323,57.569,160.498
C04822=1013.434,128.233,-124.379,166.320,57.581,160.499
C04823=1013.430,127.984,-124.362,166.317,57.592,160.501
C04824=1013.425,127.734,-124.344,166.315,57.603,160.503
C04825=1013.421,127.485,-124.327,166.311,57.615,160.504
C04826=1013.417,127.236,-124.310,166.309,57.626,160.506
C04827=1013.412,126.986,-124.292,166.306,57.637,160.507
C04828=1013.409,126.737,-124.275,166.303,57.649,160.509
C04829=1013.405,126.488,-124.258,166.300,57.660,160.510
C04830=1013.400,126.239,-124.240,166.297,57.672,160.512
C04831=1013.396,125.989,-124.223,166.295,57.683,160.513
C04832=1013.392,125.739,-124.205,166.292,57.695,160.515
C04833=1013.388,125.490,-124.188,166.288,57.706,160.516
C04834=1013.384,125.241,-124.170,166.286,57.717,160.518
C04835=1013.380,124.991,-124.152,166.283,57.729,160.519
C04836=1013.376,124.742,-124.135,166.281,57.740,160.521
C04837=1013.372,124.493,-124.118,166.278,57.751,160.523
C04838=1013.367,124.243,-124.100,166.276,57.763,160.524
C04839=1013.363,123.994,-124.083,166.272,57.774,160.526
C04840=1013.360,123.745,-124.066,166.270,57.785,160.527
C04841=1013.355,123.495,-124.048,166.267,57.797,160.529
C04842=1013.351,123.246,-124.030,166.264,57.808,160.530
C04843=1013.347,122.997,-124.013,166.262,57.820,160.532
C04844=1013.342,122.717,-123.994,166.259,57.832,160.534
C04845=1013.338,122.437,-123.975,166.255,57.845,160.536
C04846=1013.333,122.158,-123.956,166.252,57.857,160.537
C04847=1013.329,121.878,-123.936,166.249,57.870,160.539
C04848=1013.324,121.628,-123.918,166.247,57.881,160.540
C04849=1013.320,121.378,-123.901,166.243,57.892,160.542
C04850=1013.316,121.129,-123.884,166.241,57.903,160.544
C04851=1013.312,120.881,-123.866,166.238,57.915,160.545
C04852=1013.308,120.631,-123.849,166.236,57.925,160.547
C04853=1013.304,120.381,-123.832,166.234,57.937,160.548
C04854=1013.300,120.132,-123.815,166.230,57.948,160.550
C04855=1013.296,119.883,-123.798,166.228,57.959,160.551
C04856=1013.292,119.633,-123.780,166.224,57.970,160.553
C04857=1013.288,119.384,-123.763,166.222,57.981,160.554
C04858=1013.284,119.135,-123.745,166.220,57.993,160.556
C04859=1013.280,118.886,-123.728,166.217,58.004,160.557
C04860=1013.275,118.636,-123.711,166.214,58.015,160.559
C04861=1013.271,118.386,-123.694,166.212,58.026,160.560
C04862=1013.268,118.137,-123.677,166.209,58.037,160.562
C04863=1013.264,117.888,-123.660,166.206,58.048,160.563
C04864=1013.259,117.638,-123.642,166.205,58.059,160.565
C04865=1013.255,117.389,-123.625,166.202,58.070,160.567
C04866=1013.251,117.139,-123.608,166.199,58.081,160.568
C04867=1013.248,116.890,-123.591,166.196,58.092,160.570
C04868=1013.243,116.641,-123.573,166.194,58.103,160.571
C04869=1013.239,116.391,-123.556,166.191,58.114,160.573
C04870=1013.235,116.142,-123.539,166.188,58.125,160.574
C04871=1013.231,115.893,-123.521,166.186,58.136,160.576
C04872=1013.227,115.644,-123.504,166.184,58.147,160.577
C04873=1013.223,115.394,-123.487,166.181,58.158,160.579
C04874=1013.219,115.144,-123.470,166.178,58.169,160.580
C04875=1013.215,114.895,-123.453,166.175,58.180,160.582
C04876=1013.211,114.646,-123.436,166.173,58.191,160.583
C04877=1013.207,114.397,-123.419,166.171,58.202,160.585
C04878=1013.203,114.147,-123.402,166.168,58.212,160.586
C04879=1013.199,113.897,-123.384,166.165,58.224,160.588
C04880=1013.195,113.648,-123.367,166.163,58.235,160.589
C04881=1013.191,113.399,-123.350,166.160,58.245,160.591
C04882=1013.187,113.150,-123.333,166.158,58.256,160.592
C04883=1013.183,112.900,-123.316,166.156,58.267,160.594
C04884=1013.180,112.651,-123.299,166.154,58.278,160.596
C04885=1013.176,112.402,-123.282,166.151,58.288,160.597
C04886=1013.171,112.152,-123.264,166.147,58.300,160.598
C04887=1013.167,111.902,-123.247,166.145,58.310,160.600
C04888=1013.164,111.653,-123.230,166.143,58.321,160.601
C04889=1013.160,111.404,-123.213,166.140,58.332,160.603
C04890=1013.155,111.154,-123.197,166.138,58.343,160.604
C04891=1013.151,110.905,-123.180,166.136,58.354,160.606
C04892=1013.148,110.656,-123.163,166.134,58.365,160.608
C04893=1013.142,110.406,-123.146,166.130,58.376,160.609
C04894=1013.139,110.156,-123.130,166.128,58.387,160.611
C04895=1013.135,109.907,-123.113,166.126,58.398,160.612
C04896=1013.131,109.658,-123.096,166.123,58.409,160.614
C04897=1013.126,109.409,-123.079,166.120,58.419,160.615
C04898=1013.123,109.159,-123.063,166.118,58.430,160.617
C04899=1013.119,108.910,-123.046,166.116,58.441,160.618
C04900=1013.114,108.661,-123.029,166.114,58.452,160.620
C04901=1013.111,108.411,-123.013,166.110,58.463,160.621
C04902=1013.106,108.162,-122.996,166.108,58.474,160.623
C04903=1013.102,107.912,-122.979,166.106,58.485,160.624
C04904=1013.097,107.662,-122.963,166.104,58.496,160.626
C04905=1013.094,107.413,-122.946,166.101,58.507,160.627
C04906=1013.089,107.164,-122.930,166.099,58.517,160.629
C04907=1013.085,106.914,-122.913,166.096,58.528,160.630
C04908=1013.081,106.635,-122.895,166.094,58.540,160.632
C04909=1013.076,106.355,-122.876,166.091,58.552,160.634
C04910=1013.071,106.076,-122.858,166.088,58.564,160.635
C04911=1013.067,105.796,-122.839,166.086,58.576,160.637
C04912=1013.063,105.547,-122.822,166.082,58.587,160.639
C04913=1013.058,105.297,-122.807,166.080,58.598,160.640
C04914=1013.055,105.048,-122.790,166.078,58.609,160.642
C04915=1013.050,104.798,-122.774,166.075,58.619,160.643
C04916=1013.046,104.549,-122.757,166.073,58.630,160.645
C04917=1013.042,104.300,-122.741,166.071,58.641,160.646
C04918=1013.038,104.050,-122.724,166.068,58.651,160.647
C04919=1013.034,103.801,-122.707,166.066,58.662,160.649
C04920=1013.030,103.552,-122.691,166.065,58.673,160.651
C04921=1013.025,103.303,-122.674,166.062,58.683,160.652
C04922=1013.022,103.053,-122.658,166.060,58.694,160.654
C04923=1013.017,102.804,-122.642,166.057,58.705,160.655
C04924=1013.014,102.554,-122.625,166.055,58.715,160.657
C04925=1013.009,102.305,-122.609,166.052,58.726,160.658
C04926=1013.006,102.055,-122.592,166.050,58.736,160.659
C04927=1013.001,101.806,-122.576,166.047,58.747,160.661
C04928=1012.997,101.556,-122.560,166.045,58.758,160.663
C04929=1012.993,101.307,-122.543,166.042,58.768,160.664
C04930=1012.989,101.057,-122.527,166.040,58.779,160.666
C04931=1012.985,100.808,-122.510,166.039,58.789,160.667
C04932=1012.981,100.558,-122.494,166.036,58.800,160.669
C04933=1012.977,100.309,-122.478,166.034,58.810,160.670
C04934=1012.973,100.060,-122.461,166.031,58.821,160.672
C04935=1012.969,99.810,-122.445,166.029,58.831,160.673
C04936=1012.965,99.561,-122.428,166.027,58.842,160.674
C04937=1012.961,99.311,-122.412,166.025,58.852,160.676
C04938=1012.956,99.062,-122.395,166.022,58.862,160.677
C04939=1012.953,98.812,-122.379,166.020,58.873,160.679
C04940=1012.949,98.562,-122.363,166.017,58.884,160.680
C04941=1012.944,98.313,-122.347,166.015,58.895,160.682
C04942=1012.940,98.064,-122.331,166.013,58.904,160.683
C04943=1012.936,97.814,-122.315,166.011,58.915,160.685
C04944=1012.932,97.564,-122.299,166.008,58.926,160.686
C04945=1012.927,97.315,-122.282,166.006,58.936,160.688
C04946=1012.923,97.066,-122.267,166.004,58.947,160.689
C04947=1012.919,96.816,-122.251,166.003,58.957,160.691
C04948=1012.916,96.567,-122.235,166.000,58.967,160.692
C04949=1012.911,96.318,-122.218,165.997,58.978,160.694
C04950=1012.907,96.069,-122.203,165.995,58.989,160.695
C04951=1012.902,95.819,-122.187,165.992,58.999,160.696
C04952=1012.898,95.569,-122.171,165.991,59.009,160.698
C04953=1012.894,95.320,-122.155,165.988,59.020,160.700
C04954=1012.890,95.071,-122.138,165.986,59.030,160.701
C04955=1012.886,94.821,-122.122,165.984,59.041,160.703
C04956=1012.881,94.571,-122.107,165.982,59.051,160.704
C04957=1012.878,94.322,-122.090,165.979,59.061,160.705
C04958=1012.874,94.073,-122.075,165.977,59.071,160.707
C04959=1012.870,93.823,-122.059,165.976,59.082,160.708
C04960=1012.865,93.574,-122.043,165.973,59.092,160.710
C04961=1012.861,93.325,-122.027,165.970,59.102,160.711
C04962=1012.857,93.075,-122.010,165.969,59.112,160.713
C04963=1012.853,92.825,-121.995,165.966,59.123,160.714
C04964=1012.849,92.576,-121.979,165.965,59.133,160.716
C04965=1012.844,92.326,-121.963,165.962,59.143,160.717
C04966=1012.840,92.078,-121.947,165.959,59.153,160.718
C04967=1012.837,91.828,-121.931,165.958,59.163,160.720
C04968=1012.832,91.578,-121.915,165.955,59.174,160.721
C04969=1012.828,91.329,-121.899,165.954,59.184,160.723
C04970=1012.824,91.079,-121.883,165.951,59.194,160.724
C04971=1012.819,90.829,-121.868,165.949,59.205,160.726
C04972=1012.816,90.594,-121.853,165.946,59.214,160.727
C04973=1012.812,90.359,-121.837,165.945,59.224,160.728
C04974=1012.808,90.124,-121.823,165.943,59.233,160.730
C04975=1012.805,89.889,-121.807,165.941,59.242,160.731
C04976=1012.800,89.654,-121.792,165.939,59.252,160.732
C04977=1012.797,89.418,-121.778,165.937,59.261,160.734
C04978=1012.793,89.183,-121.763,165.935,59.270,160.735
C04979=1012.789,88.948,-121.747,165.933,59.280,160.737
C04980=1012.785,88.699,-121.732,165.931,59.291,160.738
C04981=1012.781,88.449,-121.716,165.929,59.300,160.739
C04982=1012.776,88.200,-121.700,165.926,59.311,160.741
C04983=1012.772,87.950,-121.684,165.925,59.321,160.742
C04984=1012.769,87.701,-121.670,165.922,59.331,160.744
C04985=1012.764,87.451,-121.654,165.921,59.341,160.745
C04986=1012.760,87.202,-121.638,165.918,59.351,160.746
C04987=1012.756,86.952,-121.622,165.916,59.361,160.748
C04988=1012.752,86.703,-121.607,165.914,59.371,160.749
C04989=1012.747,86.454,-121.592,165.912,59.381,160.751
C04990=1012.743,86.204,-121.576,165.911,59.391,160.752
C04991=1012.739,85.954,-121.561,165.908,59.401,160.754
C04992=1012.734,85.704,-121.545,165.906,59.411,160.755
C04993=1012.731,85.456,-121.530,165.904,59.421,160.757
C04994=1012.726,85.206,-121.514,165.902,59.430,160.758
C04995=1012.722,84.956,-121.498,165.899,59.441,160.759
C04996=1012.718,84.707,-121.482,165.897,59.451,160.761
C04997=1012.714,84.457,-121.468,165.896,59.460,160.762
C04998=1012.709,84.208,-121.453,165.893,59.471,160.764
C04999=1012.705,83.959,-121.437,165.892,59.481,160.765
C05000=1012.676,96.231,-122.618,165.960,59.184,160.725
C05001=1012.680,96.481,-122.634,165.963,59.174,160.724
C05002=1012.685,96.730,-122.650,165.965,59.164,160.722
C05003=1012.688,96.979,-122.666,165.967,59.154,160.721
C05004=1012.692,97.229,-122.682,165.969,59.143,160.719
C05005=1012.697,97.478,-122.698,165.971,59.133,160.718
C05006=1012.701,97.728,-122.713,165.974,59.123,160.716
C05007=1012.705,97.977,-122.729,165.976,59.113,160.715
C05008=1012.709,98.227,-122.746,165.979,59.102,160.713
C05009=1012.713,98.476,-122.762,165.980,59.092,160.712
C05010=1012.718,98.726,-122.778,165.983,59.082,160.711
C05011=1012.721,98.976,-122.794,165.985,59.071,160.709
C05012=1012.726,99.225,-122.811,165.987,59.061,160.707
C05013=1012.729,99.474,-122.827,165.989,59.051,160.706
C05014=1012.733,99.723,-122.842,165.992,59.040,160.705
C05015=1012.737,99.973,-122.860,165.993,59.030,160.703
C05016=1012.741,100.222,-122.875,165.996,59.020,160.702
C05017=1012.745,100.472,-122.892,165.999,59.009,160.700
C05018=1012.749,100.721,-122.908,166.000,59.000,160.699
C05019=1012.753,100.971,-122.925,166.002,58.989,160.697
C05020=1012.758,101.220,-122.941,166.005,58.978,160.696
C05021=1012.761,101.470,-122.957,166.008,58.968,160.695
C05022=1012.766,101.719,-122.974,166.009,58.958,160.693
C05023=1012.769,101.969,-122.990,166.012,58.947,160.692
C05024=1012.774,102.218,-123.006,166.014,58.936,160.690
C05025=1012.777,102.467,-123.023,166.016,58.926,160.689
C05026=1012.781,102.716,-123.038,166.019,58.916,160.687
C05027=1012.785,102.966,-123.056,166.020,58.905,160.686
C05028=1012.789,103.215,-123.071,166.023,58.895,160.684
C05029=1012.793,103.465,-123.088,166.025,58.884,160.683
C05030=1012.798,103.714,-123.104,166.028,58.874,160.681
C05031=1012.801,103.963,-123.121,166.030,58.863,160.680
C05032=1012.806,104.213,-123.137,166.033,58.853,160.678
C05033=1012.809,104.463,-123.153,166.035,58.842,160.677
C05034=1012.814,104.712,-123.170,166.038,58.832,160.676
C05035=1012.818,104.962,-123.186,166.039,58.821,160.674
C05036=1012.821,105.211,-123.203,166.041,58.810,160.672
C05037=1012.828,105.628,-123.231,166.046,58.792,160.670
C05038=1012.835,106.045,-123.258,166.049,58.774,160.667
C05039=1012.842,106.462,-123.286,166.053,58.757,160.665
C05040=1012.849,106.879,-123.313,166.058,58.739,160.662
C05041=1012.853,107.130,-123.329,166.060,58.728,160.661
C05042=1012.857,107.379,-123.346,166.063,58.718,160.659
C05043=1012.862,107.629,-123.362,166.065,58.707,160.658
C05044=1012.865,107.878,-123.379,166.067,58.696,160.656
C05045=1012.870,108.127,-123.395,166.069,58.685,160.655
C05046=1012.874,108.377,-123.412,166.072,58.675,160.653
C05047=1012.878,108.626,-123.428,166.074,58.664,160.652
C05048=1012.882,108.876,-123.445,166.076,58.653,160.650
C05049=1012.886,109.125,-123.462,166.079,58.642,160.649
C05050=1012.890,109.374,-123.478,166.081,58.632,160.647
C05051=1012.894,109.624,-123.495,166.084,58.621,160.646
C05052=1012.898,109.873,-123.512,166.086,58.610,160.644
C05053=1012.902,110.122,-123.528,166.089,58.600,160.643
C05054=1012.906,110.372,-123.545,166.091,58.589,160.641
C05055=1012.910,110.621,-123.562,166.093,58.578,160.640
C05056=1012.914,110.870,-123.578,166.095,58.567,160.638
C05057=1012.918,111.120,-123.595,166.098,58.556,160.636
C05058=1012.922,111.369,-123.612,166.101,58.545,160.635
C05059=1012.926,111.618,-123.629,166.104,58.534,160.634
C05060=1012.930,111.867,-123.645,166.106,58.524,160.632
C05061=1012.935,112.118,-123.662,166.108,58.513,160.631
C05062=1012.938,112.368,-123.680,166.110,58.502,160.629
C05063=1012.942,112.617,-123.697,166.113,58.492,160.628
C05064=1012.945,112.866,-123.714,166.116,58.481,160.626
C05065=1012.949,113.115,-123.731,166.118,58.470,160.625
C05066=1012.953,113.365,-123.748,166.120,58.459,160.623
C05067=1012.957,113.614,-123.765,166.123,58.449,160.622
C05068=1012.961,113.863,-123.782,166.125,58.438,160.620
C05069=1012.965,114.112,-123.799,166.127,58.427,160.619
C05070=1012.969,114.362,-123.816,166.130,58.416,160.617
C05071=1012.973,114.612,-123.834,166.133,58.405,160.616
C05072=1012.977,114.861,-123.851,166.135,58.394,160.614
C05073=1012.981,115.110,-123.868,166.138,58.384,160.613
C05074=1012.985,115.359,-123.885,166.140,58.373,160.611
C05075=1012.989,115.609,-123.902,166.143,58.362,160.610
C05076=1012.992,115.858,-123.919,166.145,58.351,160.608
C05077=1012.996,116.108,-123.936,166.147,58.340,160.607
C05078=1013.000,116.357,-123.953,166.151,58.329,160.605
C05079=1013.004,116.607,-123.970,166.153,58.318,160.604
C05080=1013.008,116.856,-123.987,166.155,58.307,160.602
C05081=1013.012,117.106,-124.004,166.157,58.296,160.600
C05082=1013.016,117.355,-124.021,166.161,58.285,160.599
C05083=1013.020,117.604,-124.038,166.163,58.274,160.597
C05084=1013.024,117.853,-124.055,166.165,58.263,160.596
C05085=1013.029,118.103,-124.074,166.168,58.252,160.594
C05086=1013.032,118.352,-124.091,166.171,58.241,160.593
C05087=1013.036,118.601,-124.108,166.173,58.230,160.591
C05088=1013.040,118.851,-124.125,166.176,58.219,160.590
C05089=1013.044,119.100,-124.142,166.178,58.208,160.588
C05090=1013.048,119.349,-124.159,166.181,58.197,160.587
C05091=1013.052,119.599,-124.176,166.184,58.186,160.585
C05092=1013.056,119.848,-124.194,166.186,58.175,160.583
C05093=1013.060,120.098,-124.211,166.189,58.163,160.582
C05094=1013.064,120.347,-124.228,166.191,58.153,160.581
C05095=1013.068,120.596,-124.245,166.194,58.142,160.579
C05096=1013.072,120.846,-124.262,166.197,58.130,160.578
C05097=1013.076,121.095,-124.279,166.199,58.120,160.576
C05098=1013.080,121.345,-124.296,166.203,58.108,160.575
C05099=1013.084,121.594,-124.313,166.204,58.097,160.573
C05100=1013.088,121.844,-124.331,166.207,58.086,160.571
C05101=1013.093,122.123,-124.350,166.211,58.073,160.570
C05102=1013.097,122.402,-124.370,166.213,58.061,160.568
C05103=1013.102,122.682,-124.389,166.217,58.048,160.566
C05104=1013.107,122.962,-124.409,166.219,58.035,160.564
C05105=1013.110,123.211,-124.426,166.222,58.024,160.563
C05106=1013.114,123.460,-124.443,166.225,58.013,160.562
C05107=1013.119,123.710,-124.461,166.227,58.002,160.560
C05108=1013.123,123.960,-124.478,166.230,57.991,160.558
C05109=1013.126,124.209,-124.495,166.232,57.980,160.557
C05110=1013.131,124.457,-124.513,166.235,57.968,160.555
C05111=1013.135,124.707,-124.530,166.238,57.957,160.554
C05112=1013.139,124.957,-124.547,166.241,57.946,160.552
C05113=1013.143,125.206,-124.564,166.243,57.934,160.550
C05114=1013.147,125.456,-124.582,166.246,57.923,160.549
C05115=1013.151,125.705,-124.599,166.250,57.912,160.548
C05116=1013.155,125.954,-124.616,166.252,57.900,160.546
C05117=1013.159,126.203,-124.634,166.255,57.889,160.544
C05118=1013.164,126.453,-124.651,166.257,57.877,160.543
C05119=1013.168,126.702,-124.668,166.260,57.866,160.541
C05120=1013.171,126.952,-124.685,166.263,57.855,160.540
C05121=1013.176,127.201,-124.703,166.266,57.843,160.538
C05122=1013.180,127.450,-124.720,166.269,57.832,160.537
C05123=1013.184,127.699,-124.737,166.271,57.821,160.535
C05124=1013.188,127.949,-124.755,166.274,57.809,160.534
C05125=1013.193,128.198,-124.773,166.276,57.798,160.532
C05126=1013.197,128.447,-124.790,166.280,57.787,160.530
C05127=1013.201,128.697,-124.807,166.283,57.775,160.529
C05128=1013.205,128.947,-124.824,166.285,57.764,160.527
C05129=1013.209,129.195,-124.842,166.288,57.752,160.526
C05130=1013.213,129.446,-124.860,166.292,57.741,160.524
C05131=1013.217,129.694,-124.878,166.293,57.729,160.522
C05132=1013.221,129.944,-124.895,166.297,57.718,160.521
C05133=1013.225,130.194,-124.913,166.299,57.706,160.519
C05134=1013.229,130.442,-124.931,166.302,57.695,160.518
C05135=1013.233,130.692,-124.948,166.306,57.684,160.517
C05136=1013.237,130.941,-124.967,166.308,57.672,160.515
C05137=1013.241,131.191,-124.984,166.311,57.661,160.513
C05138=1013.245,131.440,-125.002,166.313,57.650,160.512
C05139=1013.248,131.690,-125.020,166.317,57.639,160.510
C05140=1013.253,131.939,-125.038,166.320,57.627,160.509
C05141=1013.257,132.188,-125.056,166.322,57.616,160.507
C05142=1013.261,132.438,-125.074,166.325,57.604,160.505
C05143=1013.265,132.686,-125.091,166.329,57.593,160.504
C05144=1013.268,132.936,-125.109,166.331,57.581,160.502
C05145=1013.273,133.185,-125.127,166.334,57.570,160.501
C05146=1013.276,133.435,-125.145,166.337,57.558,160.499
C05147=1013.281,133.684,-125.163,166.340,57.547,160.498
C05148=1013.285,133.934,-125.180,166.343,57.535,160.496
C05149=1013.289,134.183,-125.199,166.345,57.524,160.495
C05150=1013.293,134.432,-125.217,166.348,57.513,160.493
C05151=1013.296,134.681,-125.234,166.351,57.501,160.491
C05152=1013.301,134.931,-125.253,166.355,57.490,160.490
C05153=1013.305,135.180,-125.270,166.358,57.478,160.489
C05154=1013.309,135.430,-125.288,166.360,57.467,160.487
C05155=1013.313,135.678,-125.306,166.363,57.455,160.485
C05156=1013.317,135.929,-125.324,166.366,57.443,160.484
C05157=1013.321,136.177,-125.342,166.369,57.433,160.482
C05158=1013.325,136.427,-125.361,166.372,57.421,160.481
C05159=1013.329,136.676,-125.378,166.375,57.409,160.479
C05160=1013.333,136.926,-125.397,166.378,57.398,160.478
C05161=1013.337,137.175,-125.414,166.381,57.386,160.476
C05162=1013.341,137.424,-125.433,166.384,57.375,160.475
C05163=1013.345,137.674,-125.450,166.387,57.363,160.473
C05164=1013.349,137.923,-125.469,166.390,57.351,160.471
C05165=1013.354,138.202,-125.490,166.393,57.338,160.470
C05166=1013.358,138.482,-125.509,166.396,57.326,160.468
C05167=1013.363,138.761,-125.530,166.400,57.313,160.466
C05168=1013.366,139.041,-125.551,166.403,57.300,160.465
C05169=1013.371,139.291,-125.569,166.406,57.288,160.463
C05170=1013.375,139.540,-125.587,166.410,57.277,160.461
C05171=1013.379,139.789,-125.606,166.412,57.266,160.460
C05172=1013.383,140.038,-125.624,166.415,57.254,160.458
C05173=1013.387,140.288,-125.642,166.418,57.242,160.457
C05174=1013.390,140.537,-125.661,166.422,57.231,160.455
C05175=1013.395,140.787,-125.678,166.425,57.219,160.454
C05176=1013.399,141.036,-125.697,166.428,57.207,160.452
C05177=1013.402,141.285,-125.715,166.431,57.197,160.451
C05178=1013.407,141.535,-125.734,166.434,57.185,160.449
C05179=1013.410,141.784,-125.752,166.437,57.173,160.447
C05180=1013.415,142.033,-125.770,166.440,57.161,160.446
C05181=1013.419,142.282,-125.789,166.444,57.150,160.445
C05182=1013.423,142.531,-125.807,166.447,57.138,160.443
C05183=1013.427,142.780,-125.825,166.450,57.126,160.441
C05184=1013.431,143.030,-125.844,166.453,57.114,160.440
C05185=1013.435,143.279,-125.863,166.455,57.103,160.438
C05186=1013.439,143.528,-125.880,166.459,57.092,160.437
C05187=1013.443,143.778,-125.899,166.462,57.080,160.435
C05188=1013.447,144.027,-125.918,166.465,57.068,160.434
C05189=1013.451,144.276,-125.936,166.468,57.056,160.432
C05190=1013.455,144.526,-125.954,166.471,57.045,160.430
C05191=1013.459,144.775,-125.973,166.475,57.034,160.429
C05192=1013.464,145.024,-125.991,166.478,57.022,160.427
C05193=1013.467,145.273,-126.009,166.481,57.010,160.426
C05194=1013.471,145.523,-126.028,166.484,56.998,160.424
C05195=1013.475,145.772,-126.047,166.487,56.986,160.423
C05196=1013.479,146.021,-126.065,166.491,56.975,160.421
C05197=1013.483,146.271,-126.083,166.494,56.963,160.420
C05198=1013.487,146.520,-126.102,166.497,56.952,160.418
C05199=1013.491,146.769,-126.121,166.500,56.940,160.417
C05200=1013.495,147.018,-126.140,166.504,56.928,160.415
C05201=1013.499,147.268,-126.159,166.507,56.916,160.413
C05202=1013.503,147.517,-126.177,166.509,56.906,160.412
C05203=1013.507,147.767,-126.196,166.513,56.894,160.410
C05204=1013.511,148.016,-126.215,166.516,56.882,160.409
C05205=1013.515,148.265,-126.234,166.519,56.870,160.407
C05206=1013.519,148.514,-126.252,166.522,56.858,160.406
C05207=1013.523,148.764,-126.271,166.525,56.847,160.404
C05208=1013.527,149.013,-126.289,166.529,56.835,160.403
C05209=1013.531,149.262,-126.308,166.532,56.824,160.401
C05210=1013.535,149.511,-126.327,166.535,56.812,160.400
C05211=1013.539,149.760,-126.346,166.539,56.800,160.398
C05212=1013.543,150.010,-126.365,166.542,56.788,160.396
C05213=1013.547,150.259,-126.384,166.545,56.777,160.395
C05214=1013.551,150.509,-126.403,166.548,56.765,160.393
C05215=1013.555,150.758,-126.421,166.551,56.753,160.392
C05216=1013.559,151.007,-126.441,166.556,56.741,160.390
C05217=1013.563,151.256,-126.459,166.559,56.730,160.389
C05218=1013.566,151.505,-126.478,166.563,56.718,160.388
C05219=1013.570,151.755,-126.496,166.566,56.706,160.386
C05220=1013.575,152.004,-126.516,166.569,56.695,160.384
C05221=1013.579,152.254,-126.535,166.572,56.683,160.383
C05222=1013.583,152.502,-126.554,166.576,56.671,160.381
C05223=1013.587,152.752,-126.573,166.579,56.659,160.380
C05224=1013.591,153.001,-126.591,166.582,56.648,160.378
C05225=1013.595,153.250,-126.611,166.585,56.636,160.377
C05226=1013.599,153.500,-126.630,166.589,56.624,160.375
C05227=1013.603,153.748,-126.649,166.592,56.612,160.373
C05228=1013.607,153.998,-126.667,166.595,56.601,160.372
C05229=1013.611,154.278,-126.689,166.600,56.587,160.370
C05230=1013.615,154.557,-126.711,166.604,56.574,160.369
C05231=1013.621,154.837,-126.732,166.607,56.562,160.367
C05232=1013.625,155.116,-126.753,166.610,56.548,160.365
C05233=1013.629,155.365,-126.773,166.614,56.536,160.363
C05234=1013.633,155.615,-126.791,166.618,56.524,160.362
C05235=1013.637,155.864,-126.811,166.621,56.512,160.361
C05236=1013.641,156.114,-126.830,166.625,56.501,160.359
C05237=1013.646,156.363,-126.849,166.628,56.489,160.357
C05238=1013.648,156.612,-126.868,166.631,56.477,160.356
C05239=1013.653,156.861,-126.887,166.635,56.465,160.354
C05240=1013.657,157.111,-126.906,166.639,56.453,160.353
C05241=1013.661,157.360,-126.926,166.642,56.442,160.351
C05242=1013.665,157.609,-126.944,166.645,56.430,160.350
C05243=1013.669,157.859,-126.964,166.649,56.418,160.348
C05244=1013.673,158.107,-126.983,166.652,56.407,160.347
C05245=1013.677,158.357,-127.002,166.655,56.395,160.345
C05246=1013.681,158.606,-127.022,166.659,56.383,160.344
C05247=1013.684,158.855,-127.042,166.664,56.372,160.343
C05248=1013.689,159.104,-127.061,166.667,56.360,160.341
C05249=1013.692,159.354,-127.081,166.670,56.348,160.339
C05250=1013.696,159.604,-127.101,166.674,56.337,160.338
C05251=1013.700,159.853,-127.120,166.677,56.325,160.336
C05252=1013.704,160.102,-127.140,166.680,56.313,160.335
C05253=1013.708,160.351,-127.160,166.684,56.302,160.333
C05254=1013.711,160.600,-127.180,166.687,56.290,160.332
C05255=1013.715,160.849,-127.200,166.691,56.279,160.330
C05256=1013.719,161.098,-127.219,166.694,56.267,160.329
C05257=1013.723,161.347,-127.239,166.699,56.255,160.328
C05258=1013.727,161.596,-127.259,166.702,56.244,160.326
C05259=1013.731,161.846,-127.279,166.705,56.232,160.324
C05260=1013.735,162.095,-127.298,166.709,56.220,160.323
C05261=1013.739,162.344,-127.318,166.712,56.209,160.321
C05262=1013.742,162.594,-127.338,166.715,56.197,160.320
C05263=1013.747,162.843,-127.358,166.719,56.185,160.318
C05264=1013.750,163.092,-127.378,166.723,56.173,160.317
C05265=1013.754,163.340,-127.397,166.727,56.161,160.315
C05266=1013.757,163.590,-127.417,166.730,56.150,160.314
C05267=1013.762,163.839,-127.436,166.733,56.138,160.312
C05268=1013.765,164.088,-127.457,166.737,56.127,160.311
C05269=1013.769,164.337,-127.477,166.741,56.114,160.309
C05270=1013.773,164.586,-127.496,166.745,56.103,160.308
C05271=1013.777,164.836,-127.516,166.748,56.091,160.306
C05272=1013.781,165.085,-127.536,166.751,56.080,160.305
C05273=1013.785,165.334,-127.556,166.756,56.067,160.303
C05274=1013.789,165.583,-127.575,166.759,56.056,160.302
C05275=1013.793,165.833,-127.595,166.763,56.044,160.300
C05276=1013.797,166.082,-127.615,166.766,56.033,160.299
C05277=1013.801,166.331,-127.635,166.770,56.021,160.297
C05278=1013.804,166.580,-127.655,166.774,56.009,160.296
C05279=1013.809,166.829,-127.674,166.777,55.997,160.294
C05280=1013.812,167.079,-127.694,166.782,55.985,160.293
C05281=1013.816,167.328,-127.714,166.785,55.974,160.291
C05282=1013.821,167.577,-127.735,166.789,55.962,160.290
C05283=1013.824,167.826,-127.755,166.793,55.950,160.289
C05284=1013.829,168.075,-127.774,166.797,55.938,160.287
C05285=1013.832,168.324,-127.794,166.800,55.927,160.286
C05286=1013.837,168.574,-127.814,166.804,55.915,160.284
C05287=1013.841,168.823,-127.834,166.808,55.903,160.283
C05288=1013.844,169.073,-127.854,166.811,55.892,160.281
C05289=1013.849,169.321,-127.874,166.816,55.880,160.280
C05290=1013.853,169.570,-127.894,166.819,55.867,160.278
C05291=1013.857,169.820,-127.914,166.822,55.856,160.276
C05292=1013.861,170.069,-127.934,166.827,55.844,160.275
C05293=1013.865,170.348,-127.956,166.831,55.831,160.273
C05294=1013.870,170.628,-127.979,166.835,55.817,160.272
C05295=1013.874,170.907,-128.002,166.839,55.804,160.270
C05296=1013.879,171.186,-128.024,166.844,55.791,160.268
C05297=1013.883,171.435,-128.044,166.847,55.779,160.267
C05298=1013.887,171.685,-128.064,166.852,55.767,160.265
C05299=1013.891,171.935,-128.084,166.855,55.755,160.264
C05300=1013.896,172.183,-128.104,166.860,55.743,160.263
C05301=1013.899,172.432,-128.124,166.863,55.731,160.261
C05302=1013.904,172.681,-128.144,166.867,55.719,160.259
C05303=1013.907,172.930,-128.165,166.871,55.708,160.258
C05304=1013.912,173.180,-128.185,166.875,55.696,160.257
C05305=1013.916,173.429,-128.204,166.879,55.684,160.255
C05306=1013.920,173.679,-128.225,166.883,55.672,160.254
C05307=1013.924,173.927,-128.245,166.886,55.660,160.252
C05308=1013.928,174.176,-128.265,166.891,55.648,160.251
C05309=1013.932,174.425,-128.284,166.894,55.636,160.249
C05310=1013.937,174.675,-128.305,166.899,55.624,160.248
C05311=1013.940,174.924,-128.325,166.903,55.613,160.246
C05312=1013.945,175.173,-128.346,166.907,55.600,160.245
C05313=1013.949,175.422,-128.366,166.910,55.589,160.243
C05314=1013.954,175.672,-128.386,166.915,55.577,160.242
C05315=1013.957,175.920,-128.406,166.918,55.565,160.240
C05316=1013.961,176.170,-128.426,166.922,55.552,160.239
C05317=1013.966,176.418,-128.447,166.926,55.541,160.237
C05318=1013.969,176.668,-128.467,166.931,55.529,160.236
C05319=1013.974,176.917,-128.487,166.935,55.517,160.234
C05320=1013.978,177.166,-128.507,166.938,55.505,160.233
C05321=1013.982,177.415,-128.527,166.943,55.493,160.231
C05322=1013.987,177.664,-128.548,166.946,55.481,160.230
C05323=1013.991,177.914,-128.568,166.951,55.469,160.228
C05324=1013.995,178.162,-128.588,166.955,55.457,160.227
C05325=1013.999,178.412,-128.608,166.959,55.445,160.225
C05326=1014.003,178.661,-128.629,166.963,55.433,160.224
C05327=1014.008,178.910,-128.649,166.966,55.421,160.222
C05328=1014.012,179.159,-128.670,166.971,55.409,160.221
C05329=1014.017,179.409,-128.689,166.976,55.397,160.219
C05330=1014.021,179.657,-128.710,166.979,55.385,160.218
C05331=1014.024,179.907,-128.730,166.983,55.373,160.216
C05332=1014.029,180.156,-128.751,166.988,55.361,160.215
C05333=1014.033,180.405,-128.771,166.991,55.350,160.214
C05334=1014.038,180.654,-128.791,166.996,55.337,160.212
C05335=1014.042,180.904,-128.812,167.000,55.325,160.211
C05336=1014.046,181.152,-128.832,167.004,55.314,160.209
C05337=1014.050,181.401,-128.852,167.008,55.301,160.207
C05338=1014.055,181.651,-128.873,167.013,55.289,160.206
C05339=1014.058,181.900,-128.894,167.016,55.278,160.205
C05340=1014.062,182.149,-128.915,167.021,55.266,160.203
C05341=1014.066,182.398,-128.936,167.025,55.254,160.202
C05342=1014.071,182.647,-128.957,167.029,55.243,160.200
C05343=1014.074,182.896,-128.979,167.033,55.231,160.199
C05344=1014.078,183.145,-129.000,167.038,55.219,160.198
C05345=1014.082,183.395,-129.021,167.041,55.208,160.196
C05346=1014.086,183.644,-129.042,167.046,55.196,160.195
C05347=1014.090,183.892,-129.063,167.050,55.184,160.193
C05348=1014.094,184.142,-129.084,167.054,55.173,160.192
C05349=1014.098,184.391,-129.105,167.058,55.161,160.190
C05350=1014.102,184.640,-129.127,167.063,55.149,160.189
C05351=1014.106,184.889,-129.147,167.067,55.137,160.188
C05352=1014.110,185.138,-129.168,167.070,55.125,160.186
C05353=1014.114,185.387,-129.189,167.075,55.113,160.185
C05354=1014.117,185.636,-129.211,167.079,55.102,160.183
